LIN {X 0,Y 143.609,Z 288.097,A -85,B 0,C 180,E1 -24488.458,E2 -24488.458} C_VEL
LIN {X 0,Y 143.503,Z 288.112,A -85,B 0,C 180,E1 -24491.628,E2 -24491.628} C_VEL
LIN {X 0,Y 143.269,Z 288.273,A -85,B 0,C 180,E1 -24497.133,E2 -24497.133} C_VEL
LIN {X 0,Y 143.376,Z 289.137,A -85,B 0,C 180,E1 -24501.358,E2 -24501.358} C_VEL
LIN {X 0,Y 143.505,Z 290.831,A -85,B 0,C 180,E1 -24508.174,E2 -24508.174} C_VEL
LIN {X 0,Y 143.599,Z 291.615,A -85,B 0,C 180,E1 -24510.634,E2 -24510.634} C_VEL
LIN {X 0,Y 144.649,Z 294.631,A -85,B 0,C 180,E1 -24511.708,E2 -24511.708} C_VEL
LIN {X 0,Y 147.147,Z 297.644,A -85,B 0,C 180,E1 -24513.694,E2 -24513.694} C_VEL
LIN {X 0,Y 149.119,Z 301.806,A -85,B 0,C 180,E1 -24515.488,E2 -24515.488} C_VEL
LIN {X 0,Y 150.527,Z 303.861,A -85,B 0,C 180,E1 -24516.55,E2 -24516.55} C_VEL
LIN {X 0,Y 154.857,Z 313.083,A -85,B 0,C 180,E1 -24520.312,E2 -24520.312} C_VEL
LIN {X 0,Y 156.952,Z 319.223,A -85,B 0,C 180,E1 -24522.467,E2 -24522.467} C_VEL
LIN {X 0,Y 158.644,Z 326.853,A -85,B 0,C 180,E1 -24524.863,E2 -24524.863} C_VEL
LIN {X 0,Y 159.712,Z 336.585,A -85,B 0,C 180,E1 -24527.852,E2 -24527.852} C_VEL
LIN {X 0,Y 159.81,Z 346.242,A -85,B 0,C 180,E1 -24530.916,E2 -24530.916} C_VEL
LIN {X 0,Y 159.176,Z 354.738,A -85,B 0,C 180,E1 -24533.821,E2 -24533.821} C_VEL
LIN {X 0,Y 158.053,Z 361.316,A -85,B 0,C 180,E1 -24536.233,E2 -24536.233} C_VEL
LIN {X 0,Y 154.42,Z 369.15,A -85,B 0,C 180,E1 -24539.203,E2 -24539.203} C_VEL
LIN {X 0,Y 151.191,Z 375.693,A -85,B 0,C 180,E1 -24542.301,E2 -24542.301} C_VEL
LIN {X 0,Y 148.829,Z 380.197,A -85,B 0,C 180,E1 -24544.85,E2 -24544.85} C_VEL
LIN {X 0,Y 145.799,Z 385.692,A -85,B 0,C 180,E1 -24548.807,E2 -24548.807} C_VEL
LIN {X 0,Y 143.393,Z 390.021,A -85,B 0,C 180,E1 -24552.898,E2 -24552.898} C_VEL
LIN {X 0,Y 142.297,Z 392.395,A -85,B 0,C 180,E1 -24555.703,E2 -24555.703} C_VEL
LIN {X 0,Y 141.459,Z 394.201,A -85,B 0,C 180,E1 -24558.538,E2 -24558.538} C_VEL
LIN {X 0,Y 140.648,Z 396.664,A -85,B 0,C 180,E1 -24564.265,E2 -24564.265} C_VEL
LIN {X 0,Y 140.521,Z 397.259,A -85,B 0,C 180,E1 -24567.133,E2 -24567.133} C_VEL
LIN {X 0,Y 140.592,Z 397.419,A -85,B 0,C 180,E1 -24570,E2 -24570} C_VEL
LIN {X 0,Y 140.521,Z 397.259,A -85,B 0,C 180,E1 -24572.867,E2 -24572.867} C_VEL
LIN {X 0,Y 140.649,Z 396.664,A -85,B 0,C 180,E1 -24575.735,E2 -24575.735} C_VEL
LIN {X 0,Y 141.461,Z 394.201,A -85,B 0,C 180,E1 -24581.462,E2 -24581.462} C_VEL
LIN {X 0,Y 142.833,Z 391.242,A -85,B 0,C 180,E1 -24585.701,E2 -24585.701} C_VEL
LIN {X 0,Y 144.926,Z 387.247,A -85,B 0,C 180,E1 -24589.843,E2 -24589.843} C_VEL
LIN {X 0,Y 147.714,Z 382.113,A -85,B 0,C 180,E1 -24593.854,E2 -24593.854} C_VEL
LIN {X 0,Y 150.6,Z 376.85,A -85,B 0,C 180,E1 -24597.064,E2 -24597.064} C_VEL
LIN {X 0,Y 153.688,Z 370.526,A -85,B 0,C 180,E1 -24600.199,E2 -24600.199} C_VEL
LIN {X 0,Y 156.598,Z 364.574,A -85,B 0,C 180,E1 -24602.584,E2 -24602.584} C_VEL
LIN {X 0,Y 158.009,Z 361.314,A -85,B 0,C 180,E1 -24603.778,E2 -24603.778} C_VEL
LIN {X 0,Y 159.397,Z 352.982,A -85,B 0,C 180,E1 -24606.827,E2 -24606.827} C_VEL
LIN {X 0,Y 159.88,Z 342.962,A -85,B 0,C 180,E1 -24610.152,E2 -24610.152} C_VEL
LIN {X 0,Y 159.446,Z 333.125,A -85,B 0,C 180,E1 -24613.193,E2 -24613.193} C_VEL
LIN {X 0,Y 158.147,Z 324.133,A -85,B 0,C 180,E1 -24615.96,E2 -24615.96} C_VEL
LIN {X 0,Y 156.268,Z 316.945,A -85,B 0,C 180,E1 -24618.337,E2 -24618.337} C_VEL
LIN {X 0,Y 152.976,Z 308.875,A -85,B 0,C 180,E1 -24621.352,E2 -24621.352} C_VEL
LIN {X 0,Y 150.448,Z 303.601,A -85,B 0,C 180,E1 -24623.532,E2 -24623.532} C_VEL
LIN {X 0,Y 147.826,Z 299.371,A -85,B 0,C 180,E1 -24625.623,E2 -24625.623} C_VEL
LIN {X 0,Y 147.009,Z 297.41,A -85,B 0,C 180,E1 -24626.426,E2 -24626.426} C_VEL
LIN {X 0,Y 144.656,Z 294.581,A -85,B 0,C 180,E1 -24628.293,E2 -24628.293} C_VEL
LIN {X 0,Y 143.65,Z 291.95,A -85,B 0,C 180,E1 -24629.276,E2 -24629.276} C_VEL
LIN {X 0,Y 143.554,Z 291.417,A -85,B 0,C 180,E1 -24629.466,E2 -24629.466} C_VEL
LIN {X 0,Y 142.735,Z 290.904,A -85,B 0,C 180,E1 -24631.797,E2 -24631.797} C_VEL
LIN {X 0,Y 141.131,Z 290.55,A -85,B 0,C 180,E1 -24634.102,E2 -24634.102} C_VEL
LIN {X 0,Y 136.638,Z 289.817,A -85,B 0,C 180,E1 -24640.45,E2 -24640.45} C_VEL
LIN {X 0,Y 136.251,Z 289.554,A -85,B 0,C 180,E1 -24642.123,E2 -24642.123} C_VEL
LIN {X 0,Y 136.231,Z 289.039,A -85,B 0,C 180,E1 -24645.035,E2 -24645.035} C_VEL
LIN {X 0,Y 136.431,Z 288.991,A -85,B 0,C 180,E1 -24648.162,E2 -24648.162} C_VEL
LIN {X 0,Y 136.548,Z 288.976,A -85,B 0,C 180,E1 -24651.101,E2 -24651.101} C_VEL
LIN {X 0,Y 137.108,Z 288.873,A -85,B 0,C 180,E1 -24659.983,E2 -24659.983} C_VEL
LIN {X 0,Y 136.538,Z 288.969,A -85,B 0,C 180,E1 -24668.865,E2 -24668.865} C_VEL
LIN {X 0,Y 136.403,Z 288.993,A -85,B 0,C 180,E1 -24671.875,E2 -24671.875} C_VEL
LIN {X 0,Y 136.155,Z 289.024,A -85,B 0,C 180,E1 -24678.022,E2 -24678.022} C_VEL
LIN {X 0,Y 136.139,Z 289.023,A -85,B 0,C 180,E1 -24681.688,E2 -24681.688} C_VEL
LIN {X 0,Y 136.07,Z 289.034,A -85,B 0,C 180,E1 -24684.996,E2 -24684.996} C_VEL
LIN {X 0,Y 136.754,Z 291.283,A -85,B 0,C 180,E1 -24685.983,E2 -24685.983} C_VEL
LIN {X 0,Y 138.867,Z 293.818,A -85,B 0,C 180,E1 -24688.285,E2 -24688.285} C_VEL
LIN {X 0,Y 140.11,Z 294.726,A -85,B 0,C 180,E1 -24689.425,E2 -24689.425} C_VEL
LIN {X 0,Y 141.489,Z 297.604,A -85,B 0,C 180,E1 -24690.999,E2 -24690.999} C_VEL
LIN {X 0,Y 143.661,Z 299.964,A -85,B 0,C 180,E1 -24692.878,E2 -24692.878} C_VEL
LIN {X 0,Y 144.804,Z 302.24,A -85,B 0,C 180,E1 -24694.074,E2 -24694.074} C_VEL
LIN {X 0,Y 146.114,Z 303.884,A -85,B 0,C 180,E1 -24695.231,E2 -24695.231} C_VEL
LIN {X 0,Y 150.59,Z 311.718,A -85,B 0,C 180,E1 -24699.357,E2 -24699.357} C_VEL
LIN {X 0,Y 154.643,Z 320.363,A -85,B 0,C 180,E1 -24703.353,E2 -24703.353} C_VEL
LIN {X 0,Y 157.904,Z 329.461,A -85,B 0,C 180,E1 -24707.206,E2 -24707.206} C_VEL
LIN {X 0,Y 160.004,Z 337.281,A -85,B 0,C 180,E1 -24710.402,E2 -24710.402} C_VEL
LIN {X 0,Y 161.566,Z 346.214,A -85,B 0,C 180,E1 -24714.116,E2 -24714.116} C_VEL
LIN {X 0,Y 162.581,Z 353.438,A -85,B 0,C 180,E1 -24717.342,E2 -24717.342} C_VEL
LIN {X 0,Y 164.624,Z 361.086,A -85,B 0,C 180,E1 -24721.391,E2 -24721.391} C_VEL
LIN {X 0,Y 167.724,Z 367.177,A -85,B 0,C 180,E1 -24725.228,E2 -24725.228} C_VEL
LIN {X 0,Y 170.999,Z 371.462,A -85,B 0,C 180,E1 -24728.291,E2 -24728.291} C_VEL
LIN {X 0,Y 176.78,Z 376.47,A -85,B 0,C 180,E1 -24732.525,E2 -24732.525} C_VEL
LIN {X 0,Y 184.262,Z 380.618,A -85,B 0,C 180,E1 -24736.771,E2 -24736.771} C_VEL
LIN {X 0,Y 192.326,Z 383.551,A -85,B 0,C 180,E1 -24740.527,E2 -24740.527} C_VEL
LIN {X 0,Y 200.968,Z 385.523,A -85,B 0,C 180,E1 -24743.978,E2 -24743.978} C_VEL
LIN {X 0,Y 206.73,Z 386.382,A -85,B 0,C 180,E1 -24746.101,E2 -24746.101} C_VEL
LIN {X 0,Y 212.196,Z 386.787,A -85,B 0,C 180,E1 -24748.102,E2 -24748.102} C_VEL
LIN {X 0,Y 216.474,Z 386.827,A -85,B 0,C 180,E1 -24750,E2 -24750} C_VEL
LIN {X 0,Y 212.23,Z 386.786,A -85,B 0,C 180,E1 -24751.898,E2 -24751.898} C_VEL
LIN {X 0,Y 204.461,Z 386.098,A -85,B 0,C 180,E1 -24754.751,E2 -24754.751} C_VEL
LIN {X 0,Y 195.201,Z 384.349,A -85,B 0,C 180,E1 -24758.28,E2 -24758.28} C_VEL
LIN {X 0,Y 186.757,Z 381.669,A -85,B 0,C 180,E1 -24762.001,E2 -24762.001} C_VEL
LIN {X 0,Y 179.348,Z 378.066,A -85,B 0,C 180,E1 -24765.92,E2 -24765.92} C_VEL
LIN {X 0,Y 173.658,Z 374.035,A -85,B 0,C 180,E1 -24769.599,E2 -24769.599} C_VEL
LIN {X 0,Y 169.332,Z 369.44,A -85,B 0,C 180,E1 -24773.186,E2 -24773.186} C_VEL
LIN {X 0,Y 165.748,Z 363.566,A -85,B 0,C 180,E1 -24777.11,E2 -24777.11} C_VEL
LIN {X 0,Y 163.445,Z 357.24,A -85,B 0,C 180,E1 -24780.72,E2 -24780.72} C_VEL
LIN {X 0,Y 161.991,Z 349.766,A -85,B 0,C 180,E1 -24784.333,E2 -24784.333} C_VEL
LIN {X 0,Y 161.21,Z 343.695,A -85,B 0,C 180,E1 -24786.941,E2 -24786.941} C_VEL
LIN {X 0,Y 159.262,Z 334.483,A -85,B 0,C 180,E1 -24790.725,E2 -24790.725} C_VEL
LIN {X 0,Y 156.773,Z 326.032,A -85,B 0,C 180,E1 -24794.196,E2 -24794.196} C_VEL
LIN {X 0,Y 153.671,Z 318.238,A -85,B 0,C 180,E1 -24797.603,E2 -24797.603} C_VEL
LIN {X 0,Y 149.725,Z 310.274,A -85,B 0,C 180,E1 -24801.43,E2 -24801.43} C_VEL
LIN {X 0,Y 145.785,Z 303.546,A -85,B 0,C 180,E1 -24805.037,E2 -24805.037} C_VEL
LIN {X 0,Y 143.651,Z 300.008,A -85,B 0,C 180,E1 -24807.119,E2 -24807.119} C_VEL
LIN {X 0,Y 142.976,Z 299.168,A -85,B 0,C 180,E1 -24807.707,E2 -24807.707} C_VEL
LIN {X 0,Y 140.831,Z 296.559,A -85,B 0,C 180,E1 -24809.672,E2 -24809.672} C_VEL
LIN {X 0,Y 140.049,Z 294.565,A -85,B 0,C 180,E1 -24810.654,E2 -24810.654} C_VEL
LIN {X 0,Y 137.336,Z 292.246,A -85,B 0,C 180,E1 -24813.318,E2 -24813.318} C_VEL
LIN {X 0,Y 136.23,Z 289.93,A -85,B 0,C 180,E1 -24814.729,E2 -24814.729} C_VEL
LIN {X 0,Y 136.041,Z 289.029,A -85,B 0,C 180,E1 -24815.202,E2 -24815.202} C_VEL
LIN {X 0,Y 136.175,Z 289.015,A -85,B 0,C 180,E1 -24818.842,E2 -24818.842} C_VEL
LIN {X 0,Y 136.217,Z 289.007,A -85,B 0,C 180,E1 -24825.069,E2 -24825.069} C_VEL
LIN {X 0,Y 136.415,Z 288.991,A -85,B 0,C 180,E1 -24828.195,E2 -24828.195} C_VEL
LIN {X 0,Y 136.538,Z 288.969,A -85,B 0,C 180,E1 -24831.135,E2 -24831.135} C_VEL
LIN {X 0,Y 137.108,Z 288.873,A -85,B 0,C 180,E1 -24840.017,E2 -24840.017} C_VEL
LIN {X 0,Y 136.539,Z 288.977,A -85,B 0,C 180,E1 -24848.9,E2 -24848.9} C_VEL
LIN {X 0,Y 136.419,Z 288.995,A -85,B 0,C 180,E1 -24851.909,E2 -24851.909} C_VEL
LIN {X 0,Y 136.231,Z 289.039,A -85,B 0,C 180,E1 -24854.965,E2 -24854.965} C_VEL
LIN {X 0,Y 136.374,Z 290.211,A -85,B 0,C 180,E1 -24861.163,E2 -24861.163} C_VEL
LIN {X 0,Y 136.392,Z 291.281,A -85,B 0,C 180,E1 -24865.073,E2 -24865.073} C_VEL
LIN {X 0,Y 137.476,Z 294.259,A -85,B 0,C 180,E1 -24866.486,E2 -24866.486} C_VEL
LIN {X 0,Y 140.055,Z 297.363,A -85,B 0,C 180,E1 -24869.082,E2 -24869.082} C_VEL
LIN {X 0,Y 140.587,Z 298.2,A -85,B 0,C 180,E1 -24869.635,E2 -24869.635} C_VEL
LIN {X 0,Y 142.177,Z 301.62,A -85,B 0,C 180,E1 -24871.388,E2 -24871.388} C_VEL
LIN {X 0,Y 143.918,Z 303.998,A -85,B 0,C 180,E1 -24872.924,E2 -24872.924} C_VEL
LIN {X 0,Y 145.548,Z 307.451,A -85,B 0,C 180,E1 -24874.584,E2 -24874.584} C_VEL
LIN {X 0,Y 146.283,Z 308.544,A -85,B 0,C 180,E1 -24875.241,E2 -24875.241} C_VEL
LIN {X 0,Y 150.363,Z 318.156,A -85,B 0,C 180,E1 -24879.449,E2 -24879.449} C_VEL
LIN {X 0,Y 152.322,Z 325.052,A -85,B 0,C 180,E1 -24882.01,E2 -24882.01} C_VEL
LIN {X 0,Y 153.319,Z 332.074,A -85,B 0,C 180,E1 -24884.393,E2 -24884.393} C_VEL
LIN {X 0,Y 153.836,Z 339.832,A -85,B 0,C 180,E1 -24886.986,E2 -24886.986} C_VEL
LIN {X 0,Y 153.724,Z 347.362,A -85,B 0,C 180,E1 -24889.557,E2 -24889.557} C_VEL
LIN {X 0,Y 152.974,Z 355.099,A -85,B 0,C 180,E1 -24892.355,E2 -24892.355} C_VEL
LIN {X 0,Y 151.982,Z 361.096,A -85,B 0,C 180,E1 -24894.689,E2 -24894.689} C_VEL
LIN {X 0,Y 150.647,Z 364.362,A -85,B 0,C 180,E1 -24895.957,E2 -24895.957} C_VEL
LIN {X 0,Y 147.618,Z 370.315,A -85,B 0,C 180,E1 -24898.42,E2 -24898.42} C_VEL
LIN {X 0,Y 144.899,Z 375.481,A -85,B 0,C 180,E1 -24900.986,E2 -24900.986} C_VEL
LIN {X 0,Y 142.43,Z 379.986,A -85,B 0,C 180,E1 -24903.635,E2 -24903.635} C_VEL
LIN {X 0,Y 139.178,Z 385.48,A -85,B 0,C 180,E1 -24907.746,E2 -24907.746} C_VEL
LIN {X 0,Y 136.585,Z 389.808,A -85,B 0,C 180,E1 -24912.018,E2 -24912.018} C_VEL
LIN {X 0,Y 135.407,Z 392.183,A -85,B 0,C 180,E1 -24914.959,E2 -24914.959} C_VEL
LIN {X 0,Y 134.493,Z 393.989,A -85,B 0,C 180,E1 -24917.935,E2 -24917.935} C_VEL
LIN {X 0,Y 133.574,Z 396.453,A -85,B 0,C 180,E1 -24923.96,E2 -24923.96} C_VEL
LIN {X 0,Y 133.433,Z 397.048,A -85,B 0,C 180,E1 -24926.981,E2 -24926.981} C_VEL
LIN {X 0,Y 133.506,Z 397.208,A -85,B 0,C 180,E1 -24930,E2 -24930} C_VEL
LIN {X 0,Y 133.433,Z 397.048,A -85,B 0,C 180,E1 -24933.019,E2 -24933.019} C_VEL
LIN {X 0,Y 133.575,Z 396.453,A -85,B 0,C 180,E1 -24936.04,E2 -24936.04} C_VEL
LIN {X 0,Y 134.494,Z 393.989,A -85,B 0,C 180,E1 -24942.065,E2 -24942.065} C_VEL
LIN {X 0,Y 135.965,Z 391.029,A -85,B 0,C 180,E1 -24946.516,E2 -24946.516} C_VEL
LIN {X 0,Y 138.231,Z 387.035,A -85,B 0,C 180,E1 -24950.848,E2 -24950.848} C_VEL
LIN {X 0,Y 141.221,Z 381.901,A -85,B 0,C 180,E1 -24955.024,E2 -24955.024} C_VEL
LIN {X 0,Y 144.271,Z 376.638,A -85,B 0,C 180,E1 -24958.356,E2 -24958.356} C_VEL
LIN {X 0,Y 147.56,Z 370.313,A -85,B 0,C 180,E1 -24961.594,E2 -24961.594} C_VEL
LIN {X 0,Y 150.628,Z 364.361,A -85,B 0,C 180,E1 -24964.048,E2 -24964.048} C_VEL
LIN {X 0,Y 151.93,Z 361.094,A -85,B 0,C 180,E1 -24965.325,E2 -24965.325} C_VEL
LIN {X 0,Y 153.353,Z 352.09,A -85,B 0,C 180,E1 -24968.802,E2 -24968.802} C_VEL
LIN {X 0,Y 153.854,Z 343.276,A -85,B 0,C 180,E1 -24971.895,E2 -24971.895} C_VEL
LIN {X 0,Y 153.634,Z 334.642,A -85,B 0,C 180,E1 -24974.768,E2 -24974.768} C_VEL
LIN {X 0,Y 152.318,Z 325.064,A -85,B 0,C 180,E1 -24977.988,E2 -24977.988} C_VEL
LIN {X 0,Y 150.344,Z 318.211,A -85,B 0,C 180,E1 -24980.545,E2 -24980.545} C_VEL
LIN {X 0,Y 146.285,Z 308.46,A -85,B 0,C 180,E1 -24984.777,E2 -24984.777} C_VEL
LIN {X 0,Y 144.151,Z 304.62,A -85,B 0,C 180,E1 -24986.824,E2 -24986.824} C_VEL
LIN {X 0,Y 143.395,Z 303.067,A -85,B 0,C 180,E1 -24987.567,E2 -24987.567} C_VEL
LIN {X 0,Y 141.188,Z 299.854,A -85,B 0,C 180,E1 -24989.615,E2 -24989.615} C_VEL
LIN {X 0,Y 140.194,Z 297.359,A -85,B 0,C 180,E1 -24990.818,E2 -24990.818} C_VEL
LIN {X 0,Y 137.634,Z 294.521,A -85,B 0,C 180,E1 -24993.342,E2 -24993.342} C_VEL
LIN {X 0,Y 136.427,Z 291.563,A -85,B 0,C 180,E1 -24994.832,E2 -24994.832} C_VEL
LIN {X 0,Y 136.332,Z 291.011,A -85,B 0,C 180,E1 -24995.119,E2 -24995.119} C_VEL
LIN {X 0,Y 136.354,Z 290.191,A -85,B 0,C 180,E1 -24998.834,E2 -24998.834} C_VEL
LIN {X 0,Y 136.251,Z 289.554,A -85,B 0,C 180,E1 -25002.123,E2 -25002.123} C_VEL
LIN {X 0,Y 135.484,Z 289.308,A -85,B 0,C 180,E1 -25004.591,E2 -25004.591} C_VEL
LIN {X 0,Y 133.912,Z 289.346,A -85,B 0,C 180,E1 -25007.034,E2 -25007.034} C_VEL
LIN {X 0,Y 129.712,Z 289.828,A -85,B 0,C 180,E1 -25013.779,E2 -25013.779} C_VEL
LIN {X 0,Y 129.514,Z 289.847,A -85,B 0,C 180,E1 -25015.551,E2 -25015.551} C_VEL
LIN {X 0,Y 130.064,Z 289.748,A -85,B 0,C 180,E1 -25019.982,E2 -25019.982} C_VEL
LIN {X 0,Y 129.461,Z 289.849,A -85,B 0,C 180,E1 -25029.354,E2 -25029.354} C_VEL
LIN {X 0,Y 129.287,Z 289.881,A -85,B 0,C 180,E1 -25032.539,E2 -25032.539} C_VEL
LIN {X 0,Y 129.105,Z 289.967,A -85,B 0,C 180,E1 -25037.299,E2 -25037.299} C_VEL
LIN {X 0,Y 129.848,Z 292.328,A -85,B 0,C 180,E1 -25038.93,E2 -25038.93} C_VEL
LIN {X 0,Y 132.279,Z 295.025,A -85,B 0,C 180,E1 -25042.63,E2 -25042.63} C_VEL
LIN {X 0,Y 133.396,Z 295.75,A -85,B 0,C 180,E1 -25043.975,E2 -25043.975} C_VEL
LIN {X 0,Y 134.673,Z 298.541,A -85,B 0,C 180,E1 -25045.895,E2 -25045.895} C_VEL
LIN {X 0,Y 136.239,Z 300.245,A -85,B 0,C 180,E1 -25047.642,E2 -25047.642} C_VEL
LIN {X 0,Y 138.58,Z 303.972,A -85,B 0,C 180,E1 -25050.452,E2 -25050.452} C_VEL
LIN {X 0,Y 139.928,Z 305.471,A -85,B 0,C 180,E1 -25051.806,E2 -25051.806} C_VEL
LIN {X 0,Y 144.316,Z 313.327,A -85,B 0,C 180,E1 -25056.601,E2 -25056.601} C_VEL
LIN {X 0,Y 147.88,Z 320.664,A -85,B 0,C 180,E1 -25060.502,E2 -25060.502} C_VEL
LIN {X 0,Y 150.909,Z 328.553,A -85,B 0,C 180,E1 -25064.287,E2 -25064.287} C_VEL
LIN {X 0,Y 153.283,Z 337.095,A -85,B 0,C 180,E1 -25068.126,E2 -25068.126} C_VEL
LIN {X 0,Y 154.911,Z 345.903,A -85,B 0,C 180,E1 -25072.069,E2 -25072.069} C_VEL
LIN {X 0,Y 155.786,Z 354.23,A -85,B 0,C 180,E1 -25075.996,E2 -25075.996} C_VEL
LIN {X 0,Y 157.254,Z 361.31,A -85,B 0,C 180,E1 -25079.901,E2 -25079.901} C_VEL
LIN {X 0,Y 159.753,Z 367.44,A -85,B 0,C 180,E1 -25083.901,E2 -25083.901} C_VEL
LIN {X 0,Y 164.072,Z 373.302,A -85,B 0,C 180,E1 -25088.477,E2 -25088.477} C_VEL
LIN {X 0,Y 169.352,Z 377.735,A -85,B 0,C 180,E1 -25092.589,E2 -25092.589} C_VEL
LIN {X 0,Y 174.91,Z 380.899,A -85,B 0,C 180,E1 -25096.05,E2 -25096.05} C_VEL
LIN {X 0,Y 180.125,Z 383.033,A -85,B 0,C 180,E1 -25098.75,E2 -25098.75} C_VEL
LIN {X 0,Y 190.926,Z 385.74,A -85,B 0,C 180,E1 -25103.513,E2 -25103.513} C_VEL
LIN {X 0,Y 197.277,Z 386.662,A -85,B 0,C 180,E1 -25105.914,E2 -25105.914} C_VEL
LIN {X 0,Y 203.847,Z 387.108,A -85,B 0,C 180,E1 -25108.314,E2 -25108.314} C_VEL
LIN {X 0,Y 208.12,Z 387.071,A -85,B 0,C 180,E1 -25110,E2 -25110} C_VEL
LIN {X 0,Y 203.098,Z 387.057,A -85,B 0,C 180,E1 -25111.983,E2 -25111.983} C_VEL
LIN {X 0,Y 197.239,Z 386.655,A -85,B 0,C 180,E1 -25114.112,E2 -25114.112} C_VEL
LIN {X 0,Y 184.95,Z 384.451,A -85,B 0,C 180,E1 -25118.995,E2 -25118.995} C_VEL
LIN {X 0,Y 179.332,Z 382.769,A -85,B 0,C 180,E1 -25121.633,E2 -25121.633} C_VEL
LIN {X 0,Y 172.442,Z 379.67,A -85,B 0,C 180,E1 -25125.443,E2 -25125.443} C_VEL
LIN {X 0,Y 165.11,Z 374.402,A -85,B 0,C 180,E1 -25130.588,E2 -25130.588} C_VEL
LIN {X 0,Y 160.912,Z 369.192,A -85,B 0,C 180,E1 -25134.795,E2 -25134.795} C_VEL
LIN {X 0,Y 158.355,Z 364.34,A -85,B 0,C 180,E1 -25138.205,E2 -25138.205} C_VEL
LIN {X 0,Y 156.439,Z 357.773,A -85,B 0,C 180,E1 -25142.118,E2 -25142.118} C_VEL
LIN {X 0,Y 155.462,Z 350.999,A -85,B 0,C 180,E1 -25145.569,E2 -25145.569} C_VEL
LIN {X 0,Y 154.741,Z 344.625,A -85,B 0,C 180,E1 -25148.506,E2 -25148.506} C_VEL
LIN {X 0,Y 152.814,Z 335.311,A -85,B 0,C 180,E1 -25152.647,E2 -25152.647} C_VEL
LIN {X 0,Y 150.398,Z 327.156,A -85,B 0,C 180,E1 -25156.348,E2 -25156.348} C_VEL
LIN {X 0,Y 147.032,Z 318.853,A -85,B 0,C 180,E1 -25160.433,E2 -25160.433} C_VEL
LIN {X 0,Y 143.683,Z 312.226,A -85,B 0,C 180,E1 -25164.081,E2 -25164.081} C_VEL
LIN {X 0,Y 139.934,Z 305.448,A -85,B 0,C 180,E1 -25168.195,E2 -25168.195} C_VEL
LIN {X 0,Y 138.54,Z 303.944,A -85,B 0,C 180,E1 -25169.585,E2 -25169.585} C_VEL
LIN {X 0,Y 136.077,Z 300.076,A -85,B 0,C 180,E1 -25172.531,E2 -25172.531} C_VEL
LIN {X 0,Y 133.999,Z 297.417,A -85,B 0,C 180,E1 -25175.006,E2 -25175.006} C_VEL
LIN {X 0,Y 133.186,Z 295.525,A -85,B 0,C 180,E1 -25176.295,E2 -25176.295} C_VEL
LIN {X 0,Y 130.378,Z 293.154,A -85,B 0,C 180,E1 -25180.127,E2 -25180.127} C_VEL
LIN {X 0,Y 129.348,Z 290.98,A -85,B 0,C 180,E1 -25182.122,E2 -25182.122} C_VEL
LIN {X 0,Y 129.113,Z 289.902,A -85,B 0,C 180,E1 -25182.804,E2 -25182.804} C_VEL
LIN {X 0,Y 129.333,Z 289.875,A -85,B 0,C 180,E1 -25187.988,E2 -25187.988} C_VEL
LIN {X 0,Y 129.461,Z 289.849,A -85,B 0,C 180,E1 -25190.646,E2 -25190.646} C_VEL
LIN {X 0,Y 130.064,Z 289.748,A -85,B 0,C 180,E1 -25200.018,E2 -25200.018} C_VEL
LIN {X 0,Y 129.465,Z 289.86,A -85,B 0,C 180,E1 -25209.39,E2 -25209.39} C_VEL
LIN {X 0,Y 129.303,Z 289.88,A -85,B 0,C 180,E1 -25212.575,E2 -25212.575} C_VEL
LIN {X 0,Y 129.253,Z 290.767,A -85,B 0,C 180,E1 -25217.113,E2 -25217.113} C_VEL
LIN {X 0,Y 130.478,Z 293.968,A -85,B 0,C 180,E1 -25219.486,E2 -25219.486} C_VEL
LIN {X 0,Y 133.716,Z 297.729,A -85,B 0,C 180,E1 -25223.952,E2 -25223.952} C_VEL
LIN {X 0,Y 135.256,Z 301.356,A -85,B 0,C 180,E1 -25226.228,E2 -25226.228} C_VEL
LIN {X 0,Y 137.325,Z 304.012,A -85,B 0,C 180,E1 -25228.481,E2 -25228.481} C_VEL
LIN {X 0,Y 138.841,Z 307.408,A -85,B 0,C 180,E1 -25230.428,E2 -25230.428} C_VEL
LIN {X 0,Y 140.016,Z 309.061,A -85,B 0,C 180,E1 -25231.654,E2 -25231.654} C_VEL
LIN {X 0,Y 142.981,Z 315.704,A -85,B 0,C 180,E1 -25235.097,E2 -25235.097} C_VEL
LIN {X 0,Y 145.866,Z 323.593,A -85,B 0,C 180,E1 -25238.799,E2 -25238.799} C_VEL
LIN {X 0,Y 147.273,Z 329.995,A -85,B 0,C 180,E1 -25241.372,E2 -25241.372} C_VEL
LIN {X 0,Y 147.871,Z 337.781,A -85,B 0,C 180,E1 -25244.152,E2 -25244.152} C_VEL
LIN {X 0,Y 147.835,Z 346.044,A -85,B 0,C 180,E1 -25247.148,E2 -25247.148} C_VEL
LIN {X 0,Y 147.215,Z 353.163,A -85,B 0,C 180,E1 -25249.824,E2 -25249.824} C_VEL
LIN {X 0,Y 145.902,Z 360.872,A -85,B 0,C 180,E1 -25252.979,E2 -25252.979} C_VEL
LIN {X 0,Y 144.787,Z 364.149,A -85,B 0,C 180,E1 -25254.375,E2 -25254.375} C_VEL
LIN {X 0,Y 141.579,Z 370.103,A -85,B 0,C 180,E1 -25256.905,E2 -25256.905} C_VEL
LIN {X 0,Y 138.168,Z 376.159,A -85,B 0,C 180,E1 -25260.076,E2 -25260.076} C_VEL
LIN {X 0,Y 136.103,Z 379.775,A -85,B 0,C 180,E1 -25262.307,E2 -25262.307} C_VEL
LIN {X 0,Y 132.609,Z 385.268,A -85,B 0,C 180,E1 -25266.579,E2 -25266.579} C_VEL
LIN {X 0,Y 129.815,Z 389.596,A -85,B 0,C 180,E1 -25271.045,E2 -25271.045} C_VEL
LIN {X 0,Y 128.544,Z 391.971,A -85,B 0,C 180,E1 -25274.135,E2 -25274.135} C_VEL
LIN {X 0,Y 127.522,Z 393.777,A -85,B 0,C 180,E1 -25277.265,E2 -25277.265} C_VEL
LIN {X 0,Y 126.495,Z 396.241,A -85,B 0,C 180,E1 -25283.62,E2 -25283.62} C_VEL
LIN {X 0,Y 126.34,Z 396.837,A -85,B 0,C 180,E1 -25286.811,E2 -25286.811} C_VEL
LIN {X 0,Y 126.422,Z 396.997,A -85,B 0,C 180,E1 -25290,E2 -25290} C_VEL
LIN {X 0,Y 126.34,Z 396.837,A -85,B 0,C 180,E1 -25293.189,E2 -25293.189} C_VEL
LIN {X 0,Y 126.496,Z 396.241,A -85,B 0,C 180,E1 -25296.38,E2 -25296.38} C_VEL
LIN {X 0,Y 127.523,Z 393.777,A -85,B 0,C 180,E1 -25302.735,E2 -25302.735} C_VEL
LIN {X 0,Y 129.137,Z 390.817,A -85,B 0,C 180,E1 -25307.417,E2 -25307.417} C_VEL
LIN {X 0,Y 131.591,Z 386.823,A -85,B 0,C 180,E1 -25311.953,E2 -25311.953} C_VEL
LIN {X 0,Y 134.801,Z 381.689,A -85,B 0,C 180,E1 -25316.305,E2 -25316.305} C_VEL
LIN {X 0,Y 137.376,Z 377.582,A -85,B 0,C 180,E1 -25319.078,E2 -25319.078} C_VEL
LIN {X 0,Y 140.718,Z 371.616,A -85,B 0,C 180,E1 -25322.387,E2 -25322.387} C_VEL
LIN {X 0,Y 143.945,Z 365.776,A -85,B 0,C 180,E1 -25325.007,E2 -25325.007} C_VEL
LIN {X 0,Y 145.426,Z 362.514,A -85,B 0,C 180,E1 -25326.299,E2 -25326.299} C_VEL
LIN {X 0,Y 146.792,Z 356.036,A -85,B 0,C 180,E1 -25328.999,E2 -25328.999} C_VEL
LIN {X 0,Y 147.651,Z 348.87,A -85,B 0,C 180,E1 -25331.787,E2 -25331.787} C_VEL
LIN {X 0,Y 147.987,Z 341.341,A -85,B 0,C 180,E1 -25334.554,E2 -25334.554} C_VEL
LIN {X 0,Y 147.593,Z 332.815,A -85,B 0,C 180,E1 -25337.623,E2 -25337.623} C_VEL
LIN {X 0,Y 146.41,Z 325.59,A -85,B 0,C 180,E1 -25340.398,E2 -25340.398} C_VEL
LIN {X 0,Y 144.223,Z 318.855,A -85,B 0,C 180,E1 -25343.331,E2 -25343.331} C_VEL
LIN {X 0,Y 142.186,Z 313.663,A -85,B 0,C 180,E1 -25345.857,E2 -25345.857} C_VEL
LIN {X 0,Y 140.025,Z 309.03,A -85,B 0,C 180,E1 -25348.348,E2 -25348.348} C_VEL
LIN {X 0,Y 138.267,Z 306.32,A -85,B 0,C 180,E1 -25350.274,E2 -25350.274} C_VEL
LIN {X 0,Y 137.039,Z 303.397,A -85,B 0,C 180,E1 -25351.872,E2 -25351.872} C_VEL
LIN {X 0,Y 134.63,Z 300.257,A -85,B 0,C 180,E1 -25354.576,E2 -25354.576} C_VEL
LIN {X 0,Y 133.541,Z 297.315,A -85,B 0,C 180,E1 -25356.324,E2 -25356.324} C_VEL
LIN {X 0,Y 130.593,Z 294.17,A -85,B 0,C 180,E1 -25360.328,E2 -25360.328} C_VEL
LIN {X 0,Y 129.359,Z 291.222,A -85,B 0,C 180,E1 -25362.596,E2 -25362.596} C_VEL
LIN {X 0,Y 129.214,Z 290.494,A -85,B 0,C 180,E1 -25363.187,E2 -25363.187} C_VEL
LIN {X 0,Y 129.349,Z 289.874,A -85,B 0,C 180,E1 -25367.956,E2 -25367.956} C_VEL
LIN {X 0,Y 129.472,Z 289.859,A -85,B 0,C 180,E1 -25370.61,E2 -25370.61} C_VEL
LIN {X 0,Y 129.514,Z 289.847,A -85,B 0,C 180,E1 -25375.551,E2 -25375.551} C_VEL
LIN {X 0,Y 129.303,Z 289.986,A -85,B 0,C 180,E1 -25377.285,E2 -25377.285} C_VEL
LIN {X 0,Y 128.604,Z 290.373,A -85,B 0,C 180,E1 -25378.998,E2 -25378.998} C_VEL
LIN {X 0,Y 126.477,Z 291.631,A -85,B 0,C 180,E1 -25382.397,E2 -25382.397} C_VEL
LIN {X 0,Y 124.5,Z 293.183,A -85,B 0,C 180,E1 -25385.908,E2 -25385.908} C_VEL
LIN {X 0,Y 124.004,Z 294.266,A -85,B 0,C 180,E1 -25388.629,E2 -25388.629} C_VEL
LIN {X 0,Y 124.153,Z 294.573,A -85,B 0,C 180,E1 -25389.542,E2 -25389.542} C_VEL
LIN {X 0,Y 126.945,Z 296.876,A -85,B 0,C 180,E1 -25396.463,E2 -25396.463} C_VEL
LIN {X 0,Y 127.896,Z 299.416,A -85,B 0,C 180,E1 -25398.814,E2 -25398.814} C_VEL
LIN {X 0,Y 130.063,Z 301.696,A -85,B 0,C 180,E1 -25402.204,E2 -25402.204} C_VEL
LIN {X 0,Y 134.06,Z 307.81,A -85,B 0,C 180,E1 -25408.131,E2 -25408.131} C_VEL
LIN {X 0,Y 136.387,Z 311.347,A -85,B 0,C 180,E1 -25410.995,E2 -25410.995} C_VEL
LIN {X 0,Y 140.84,Z 320.252,A -85,B 0,C 180,E1 -25416.761,E2 -25416.761} C_VEL
LIN {X 0,Y 143.729,Z 327.344,A -85,B 0,C 180,E1 -25420.753,E2 -25420.753} C_VEL
LIN {X 0,Y 145.891,Z 334.212,A -85,B 0,C 180,E1 -25424.279,E2 -25424.279} C_VEL
LIN {X 0,Y 147.422,Z 340.639,A -85,B 0,C 180,E1 -25427.431,E2 -25427.431} C_VEL
LIN {X 0,Y 148.593,Z 348.009,A -85,B 0,C 180,E1 -25431.019,E2 -25431.019} C_VEL
LIN {X 0,Y 149.122,Z 354.244,A -85,B 0,C 180,E1 -25434.131,E2 -25434.131} C_VEL
LIN {X 0,Y 150.094,Z 361.488,A -85,B 0,C 180,E1 -25438.262,E2 -25438.262} C_VEL
LIN {X 0,Y 152.049,Z 367.697,A -85,B 0,C 180,E1 -25442.47,E2 -25442.47} C_VEL
LIN {X 0,Y 154.494,Z 371.993,A -85,B 0,C 180,E1 -25445.832,E2 -25445.832} C_VEL
LIN {X 0,Y 159.495,Z 377.237,A -85,B 0,C 180,E1 -25450.765,E2 -25450.765} C_VEL
LIN {X 0,Y 165.732,Z 381.175,A -85,B 0,C 180,E1 -25455.26,E2 -25455.26} C_VEL
LIN {X 0,Y 171.908,Z 383.709,A -85,B 0,C 180,E1 -25458.776,E2 -25458.776} C_VEL
LIN {X 0,Y 177.589,Z 385.325,A -85,B 0,C 180,E1 -25461.521,E2 -25461.521} C_VEL
LIN {X 0,Y 187.645,Z 386.946,A -85,B 0,C 180,E1 -25465.704,E2 -25465.704} C_VEL
LIN {X 0,Y 196.759,Z 387.401,A -85,B 0,C 180,E1 -25469.029,E2 -25469.029} C_VEL
LIN {X 0,Y 199.347,Z 387.327,A -85,B 0,C 180,E1 -25470,E2 -25470} C_VEL
LIN {X 0,Y 193.703,Z 387.335,A -85,B 0,C 180,E1 -25472.079,E2 -25472.079} C_VEL
LIN {X 0,Y 183.639,Z 386.411,A -85,B 0,C 180,E1 -25475.87,E2 -25475.87} C_VEL
LIN {X 0,Y 176.048,Z 384.914,A -85,B 0,C 180,E1 -25479.188,E2 -25479.188} C_VEL
LIN {X 0,Y 170.663,Z 383.321,A -85,B 0,C 180,E1 -25481.882,E2 -25481.882} C_VEL
LIN {X 0,Y 161.907,Z 379.027,A -85,B 0,C 180,E1 -25487.32,E2 -25487.32} C_VEL
LIN {X 0,Y 157.572,Z 375.616,A -85,B 0,C 180,E1 -25490.904,E2 -25490.904} C_VEL
LIN {X 0,Y 153.217,Z 369.907,A -85,B 0,C 180,E1 -25495.832,E2 -25495.832} C_VEL
LIN {X 0,Y 150.752,Z 363.987,A -85,B 0,C 180,E1 -25500.118,E2 -25500.118} C_VEL
LIN {X 0,Y 149.513,Z 358.185,A -85,B 0,C 180,E1 -25503.716,E2 -25503.716} C_VEL
LIN {X 0,Y 148.831,Z 350.25,A -85,B 0,C 180,E1 -25507.869,E2 -25507.869} C_VEL
LIN {X 0,Y 147.857,Z 343.259,A -85,B 0,C 180,E1 -25511.326,E2 -25511.326} C_VEL
LIN {X 0,Y 146.343,Z 335.853,A -85,B 0,C 180,E1 -25514.926,E2 -25514.926} C_VEL
LIN {X 0,Y 144.353,Z 329.202,A -85,B 0,C 180,E1 -25518.318,E2 -25518.318} C_VEL
LIN {X 0,Y 141.15,Z 320.983,A -85,B 0,C 180,E1 -25522.811,E2 -25522.811} C_VEL
LIN {X 0,Y 138.528,Z 315.595,A -85,B 0,C 180,E1 -25526.101,E2 -25526.101} C_VEL
LIN {X 0,Y 136.393,Z 311.33,A -85,B 0,C 180,E1 -25529.006,E2 -25529.006} C_VEL
LIN {X 0,Y 132.958,Z 306.215,A -85,B 0,C 180,E1 -25533.323,E2 -25533.323} C_VEL
LIN {X 0,Y 129.794,Z 301.49,A -85,B 0,C 180,E1 -25538.166,E2 -25538.166} C_VEL
LIN {X 0,Y 127.474,Z 298.631,A -85,B 0,C 180,E1 -25542.058,E2 -25542.058} C_VEL
LIN {X 0,Y 126.775,Z 296.589,A -85,B 0,C 180,E1 -25543.928,E2 -25543.928} C_VEL
LIN {X 0,Y 123.195,Z 291.592,A -85,B 0,C 180,E1 -25560.019,E2 -25560.019} C_VEL
LIN {X 0,Y 124.226,Z 294.671,A -85,B 0,C 180,E1 -25568.969,E2 -25568.969} C_VEL
LIN {X 0,Y 127.123,Z 297.333,A -85,B 0,C 180,E1 -25576.065,E2 -25576.065} C_VEL
LIN {X 0,Y 128.333,Z 300.757,A -85,B 0,C 180,E1 -25578.993,E2 -25578.993} C_VEL
LIN {X 0,Y 130.944,Z 303.97,A -85,B 0,C 180,E1 -25582.918,E2 -25582.918} C_VEL
LIN {X 0,Y 132.194,Z 307.266,A -85,B 0,C 180,E1 -25585.188,E2 -25585.188} C_VEL
LIN {X 0,Y 133.843,Z 309.656,A -85,B 0,C 180,E1 -25587.369,E2 -25587.369} C_VEL
LIN {X 0,Y 135.336,Z 313.213,A -85,B 0,C 180,E1 -25589.578,E2 -25589.578} C_VEL
LIN {X 0,Y 136.49,Z 315.349,A -85,B 0,C 180,E1 -25591.009,E2 -25591.009} C_VEL
LIN {X 0,Y 138.489,Z 320.43,A -85,B 0,C 180,E1 -25593.951,E2 -25593.951} C_VEL
LIN {X 0,Y 140.9,Z 327.821,A -85,B 0,C 180,E1 -25597.682,E2 -25597.682} C_VEL
LIN {X 0,Y 142.094,Z 335.067,A -85,B 0,C 180,E1 -25600.742,E2 -25600.742} C_VEL
LIN {X 0,Y 142.144,Z 344.465,A -85,B 0,C 180,E1 -25604.397,E2 -25604.397} C_VEL
LIN {X 0,Y 141.459,Z 352.489,A -85,B 0,C 180,E1 -25607.608,E2 -25607.608} C_VEL
LIN {X 0,Y 139.945,Z 360.647,A -85,B 0,C 180,E1 -25611.117,E2 -25611.117} C_VEL
LIN {X 0,Y 138.988,Z 363.935,A -85,B 0,C 180,E1 -25612.643,E2 -25612.643} C_VEL
LIN {X 0,Y 135.647,Z 369.89,A -85,B 0,C 180,E1 -25615.256,E2 -25615.256} C_VEL
LIN {X 0,Y 131.641,Z 376.559,A -85,B 0,C 180,E1 -25618.901,E2 -25618.901} C_VEL
LIN {X 0,Y 128.468,Z 381.477,A -85,B 0,C 180,E1 -25622.29,E2 -25622.29} C_VEL
LIN {X 0,Y 125.013,Z 386.611,A -85,B 0,C 180,E1 -25626.826,E2 -25626.826} C_VEL
LIN {X 0,Y 122.331,Z 390.604,A -85,B 0,C 180,E1 -25631.58,E2 -25631.58} C_VEL
LIN {X 0,Y 120.583,Z 393.565,A -85,B 0,C 180,E1 -25636.519,E2 -25636.519} C_VEL
LIN {X 0,Y 119.442,Z 396.029,A -85,B 0,C 180,E1 -25643.242,E2 -25643.242} C_VEL
LIN {X 0,Y 119.257,Z 396.625,A -85,B 0,C 180,E1 -25646.622,E2 -25646.622} C_VEL
LIN {X 0,Y 119.324,Z 396.786,A -85,B 0,C 180,E1 -25650,E2 -25650} C_VEL
LIN {X 0,Y 119.257,Z 396.625,A -85,B 0,C 180,E1 -25653.378,E2 -25653.378} C_VEL
LIN {X 0,Y 119.442,Z 396.029,A -85,B 0,C 180,E1 -25656.758,E2 -25656.758} C_VEL
LIN {X 0,Y 120.583,Z 393.565,A -85,B 0,C 180,E1 -25663.481,E2 -25663.481} C_VEL
LIN {X 0,Y 122.33,Z 390.604,A -85,B 0,C 180,E1 -25668.42,E2 -25668.42} C_VEL
LIN {X 0,Y 125.011,Z 386.611,A -85,B 0,C 180,E1 -25673.174,E2 -25673.174} C_VEL
LIN {X 0,Y 128.462,Z 381.477,A -85,B 0,C 180,E1 -25677.711,E2 -25677.711} C_VEL
LIN {X 0,Y 132.357,Z 375.397,A -85,B 0,C 180,E1 -25681.806,E2 -25681.806} C_VEL
LIN {X 0,Y 136.445,Z 368.512,A -85,B 0,C 180,E1 -25685.412,E2 -25685.412} C_VEL
LIN {X 0,Y 138.942,Z 363.933,A -85,B 0,C 180,E1 -25687.371,E2 -25687.371} C_VEL
LIN {X 0,Y 140.333,Z 358.874,A -85,B 0,C 180,E1 -25689.682,E2 -25689.682} C_VEL
LIN {X 0,Y 141.641,Z 350.632,A -85,B 0,C 180,E1 -25693.148,E2 -25693.148} C_VEL
LIN {X 0,Y 142.241,Z 341.6,A -85,B 0,C 180,E1 -25696.691,E2 -25696.691} C_VEL
LIN {X 0,Y 141.932,Z 333.401,A -85,B 0,C 180,E1 -25699.912,E2 -25699.912} C_VEL
LIN {X 0,Y 140.883,Z 327.86,A -85,B 0,C 180,E1 -25702.313,E2 -25702.313} C_VEL
LIN {X 0,Y 139.058,Z 321.934,A -85,B 0,C 180,E1 -25705.243,E2 -25705.243} C_VEL
LIN {X 0,Y 137.466,Z 317.859,A -85,B 0,C 180,E1 -25707.515,E2 -25707.515} C_VEL
LIN {X 0,Y 136.275,Z 314.578,A -85,B 0,C 180,E1 -25709.368,E2 -25709.368} C_VEL
LIN {X 0,Y 134.287,Z 310.947,A -85,B 0,C 180,E1 -25711.882,E2 -25711.882} C_VEL
LIN {X 0,Y 133.849,Z 309.636,A -85,B 0,C 180,E1 -25712.632,E2 -25712.632} C_VEL
LIN {X 0,Y 131.738,Z 306.306,A -85,B 0,C 180,E1 -25715.56,E2 -25715.56} C_VEL
LIN {X 0,Y 130.701,Z 303.527,A -85,B 0,C 180,E1 -25717.455,E2 -25717.455} C_VEL
LIN {X 0,Y 127.945,Z 299.982,A -85,B 0,C 180,E1 -25721.777,E2 -25721.777} C_VEL
LIN {X 0,Y 127.05,Z 297.122,A -85,B 0,C 180,E1 -25724.131,E2 -25724.131} C_VEL
LIN {X 0,Y 123.183,Z 291.609,A -85,B 0,C 180,E1 -25739.981,E2 -25739.981} C_VEL
LIN {X 0,Y 124.153,Z 294.573,A -85,B 0,C 180,E1 -25749.542,E2 -25749.542} C_VEL
LIN {X 0,Y 124.805,Z 296.181,A -85,B 0,C 180,E1 -25752.134,E2 -25752.134} C_VEL
LIN {X 0,Y 125.339,Z 298.869,A -85,B 0,C 180,E1 -25754.551,E2 -25754.551} C_VEL
LIN {X 0,Y 126.821,Z 307.274,A -85,B 0,C 180,E1 -25760.747,E2 -25760.747} C_VEL
LIN {X 0,Y 127.628,Z 308.839,A -85,B 0,C 180,E1 -25762.373,E2 -25762.373} C_VEL
LIN {X 0,Y 130.533,Z 313.591,A -85,B 0,C 180,E1 -25767.213,E2 -25767.213} C_VEL
LIN {X 0,Y 132.5,Z 317.066,A -85,B 0,C 180,E1 -25770.235,E2 -25770.235} C_VEL
LIN {X 0,Y 135.919,Z 324.614,A -85,B 0,C 180,E1 -25775.547,E2 -25775.547} C_VEL
LIN {X 0,Y 138.321,Z 330.905,A -85,B 0,C 180,E1 -25779.406,E2 -25779.406} C_VEL
LIN {X 0,Y 140.401,Z 338.193,A -85,B 0,C 180,E1 -25783.468,E2 -25783.468} C_VEL
LIN {X 0,Y 141.629,Z 344.573,A -85,B 0,C 180,E1 -25786.888,E2 -25786.888} C_VEL
LIN {X 0,Y 142.581,Z 353.267,A -85,B 0,C 180,E1 -25791.524,E2 -25791.524} C_VEL
LIN {X 0,Y 143.13,Z 361.785,A -85,B 0,C 180,E1 -25796.553,E2 -25796.553} C_VEL
LIN {X 0,Y 144.579,Z 368.072,A -85,B 0,C 180,E1 -25801.003,E2 -25801.003} C_VEL
LIN {X 0,Y 147.045,Z 373.066,A -85,B 0,C 180,E1 -25805.199,E2 -25805.199} C_VEL
LIN {X 0,Y 150.407,Z 377.048,A -85,B 0,C 180,E1 -25809.1,E2 -25809.1} C_VEL
LIN {X 0,Y 154.483,Z 380.273,A -85,B 0,C 180,E1 -25812.755,E2 -25812.755} C_VEL
LIN {X 0,Y 161.364,Z 383.605,A -85,B 0,C 180,E1 -25817.422,E2 -25817.422} C_VEL
LIN {X 0,Y 170.239,Z 386.048,A -85,B 0,C 180,E1 -25822.093,E2 -25822.093} C_VEL
LIN {X 0,Y 177.98,Z 387.23,A -85,B 0,C 180,E1 -25825.47,E2 -25825.47} C_VEL
LIN {X 0,Y 184.135,Z 387.619,A -85,B 0,C 180,E1 -25827.813,E2 -25827.813} C_VEL
LIN {X 0,Y 190.265,Z 387.592,A -85,B 0,C 180,E1 -25830,E2 -25830} C_VEL
LIN {X 0,Y 182.872,Z 387.541,A -85,B 0,C 180,E1 -25832.651,E2 -25832.651} C_VEL
LIN {X 0,Y 176.373,Z 387.069,A -85,B 0,C 180,E1 -25835.195,E2 -25835.195} C_VEL
LIN {X 0,Y 166.512,Z 385.196,A -85,B 0,C 180,E1 -25839.72,E2 -25839.72} C_VEL
LIN {X 0,Y 159.217,Z 382.704,A -85,B 0,C 180,E1 -25843.884,E2 -25843.884} C_VEL
LIN {X 0,Y 152.527,Z 378.893,A -85,B 0,C 180,E1 -25848.816,E2 -25848.816} C_VEL
LIN {X 0,Y 148.119,Z 374.452,A -85,B 0,C 180,E1 -25853.471,E2 -25853.471} C_VEL
LIN {X 0,Y 145.47,Z 370.162,A -85,B 0,C 180,E1 -25857.32,E2 -25857.32} C_VEL
LIN {X 0,Y 143.59,Z 364.308,A -85,B 0,C 180,E1 -25861.745,E2 -25861.745} C_VEL
LIN {X 0,Y 142.829,Z 358.76,A -85,B 0,C 180,E1 -25865.342,E2 -25865.342} C_VEL
LIN {X 0,Y 142.486,Z 351.903,A -85,B 0,C 180,E1 -25869.191,E2 -25869.191} C_VEL
LIN {X 0,Y 141.432,Z 343.582,A -85,B 0,C 180,E1 -25873.629,E2 -25873.629} C_VEL
LIN {X 0,Y 140.009,Z 336.642,A -85,B 0,C 180,E1 -25877.365,E2 -25877.365} C_VEL
LIN {X 0,Y 137.398,Z 328.32,A -85,B 0,C 180,E1 -25882.159,E2 -25882.159} C_VEL
LIN {X 0,Y 134.518,Z 321.325,A -85,B 0,C 180,E1 -25886.711,E2 -25886.711} C_VEL
LIN {X 0,Y 132.507,Z 317.048,A -85,B 0,C 180,E1 -25889.766,E2 -25889.766} C_VEL
LIN {X 0,Y 129.587,Z 312.102,A -85,B 0,C 180,E1 -25894.308,E2 -25894.308} C_VEL
LIN {X 0,Y 126.911,Z 307.757,A -85,B 0,C 180,E1 -25898.924,E2 -25898.924} C_VEL
LIN {X 0,Y 124.953,Z 304.943,A -85,B 0,C 180,E1 -25902.969,E2 -25902.969} C_VEL
LIN {X 0,Y 124.749,Z 304.294,A -85,B 0,C 180,E1 -25903.66,E2 -25903.66} C_VEL
LIN {X 0,Y 122.969,Z 302.161,A -85,B 0,C 180,E1 -25908.481,E2 -25908.481} C_VEL
LIN {X 0,Y 121.569,Z 298.631,A -85,B 0,C 180,E1 -25920.019,E2 -25920.019} C_VEL
LIN {X 0,Y 124.634,Z 303.64,A -85,B 0,C 180,E1 -25934.718,E2 -25934.718} C_VEL
LIN {X 0,Y 125.828,Z 307.207,A -85,B 0,C 180,E1 -25938.286,E2 -25938.286} C_VEL
LIN {X 0,Y 127.306,Z 309.327,A -85,B 0,C 180,E1 -25941.047,E2 -25941.047} C_VEL
LIN {X 0,Y 129.897,Z 314.677,A -85,B 0,C 180,E1 -25945.666,E2 -25945.666} C_VEL
LIN {X 0,Y 132.11,Z 319.814,A -85,B 0,C 180,E1 -25949.496,E2 -25949.496} C_VEL
LIN {X 0,Y 134.194,Z 325.702,A -85,B 0,C 180,E1 -25953.078,E2 -25953.078} C_VEL
LIN {X 0,Y 136.078,Z 332.93,A -85,B 0,C 180,E1 -25956.993,E2 -25956.993} C_VEL
LIN {X 0,Y 136.598,Z 338.343,A -85,B 0,C 180,E1 -25959.49,E2 -25959.49} C_VEL
LIN {X 0,Y 136.4,Z 345.808,A -85,B 0,C 180,E1 -25962.628,E2 -25962.628} C_VEL
LIN {X 0,Y 135.411,Z 354.03,A -85,B 0,C 180,E1 -25966.172,E2 -25966.172} C_VEL
LIN {X 0,Y 134.08,Z 360.42,A -85,B 0,C 180,E1 -25969.066,E2 -25969.066} C_VEL
LIN {X 0,Y 132.502,Z 365.351,A -85,B 0,C 180,E1 -25971.449,E2 -25971.449} C_VEL
LIN {X 0,Y 127.359,Z 373.686,A -85,B 0,C 180,E1 -25975.555,E2 -25975.555} C_VEL
LIN {X 0,Y 123.643,Z 379.35,A -85,B 0,C 180,E1 -25979.232,E2 -25979.232} C_VEL
LIN {X 0,Y 119.662,Z 384.844,A -85,B 0,C 180,E1 -25983.865,E2 -25983.865} C_VEL
LIN {X 0,Y 116.423,Z 389.172,A -85,B 0,C 180,E1 -25988.765,E2 -25988.765} C_VEL
LIN {X 0,Y 114.862,Z 391.546,A -85,B 0,C 180,E1 -25992.186,E2 -25992.186} C_VEL
LIN {X 0,Y 113.674,Z 393.353,A -85,B 0,C 180,E1 -25995.682,E2 -25995.682} C_VEL
LIN {X 0,Y 112.366,Z 395.817,A -85,B 0,C 180,E1 -26002.814,E2 -26002.814} C_VEL
LIN {X 0,Y 112.167,Z 396.414,A -85,B 0,C 180,E1 -26006.408,E2 -26006.408} C_VEL
LIN {X 0,Y 112.237,Z 396.575,A -85,B 0,C 180,E1 -26010,E2 -26010} C_VEL
LIN {X 0,Y 112.167,Z 396.414,A -85,B 0,C 180,E1 -26013.592,E2 -26013.592} C_VEL
LIN {X 0,Y 112.366,Z 395.817,A -85,B 0,C 180,E1 -26017.186,E2 -26017.186} C_VEL
LIN {X 0,Y 113.675,Z 393.353,A -85,B 0,C 180,E1 -26024.318,E2 -26024.318} C_VEL
LIN {X 0,Y 115.577,Z 390.392,A -85,B 0,C 180,E1 -26029.538,E2 -26029.538} C_VEL
LIN {X 0,Y 118.497,Z 386.399,A -85,B 0,C 180,E1 -26034.529,E2 -26034.529} C_VEL
LIN {X 0,Y 122.209,Z 381.265,A -85,B 0,C 180,E1 -26039.262,E2 -26039.262} C_VEL
LIN {X 0,Y 125.919,Z 375.808,A -85,B 0,C 180,E1 -26043.126,E2 -26043.126} C_VEL
LIN {X 0,Y 129.822,Z 369.677,A -85,B 0,C 180,E1 -26046.547,E2 -26046.547} C_VEL
LIN {X 0,Y 132.478,Z 365.35,A -85,B 0,C 180,E1 -26048.56,E2 -26048.56} C_VEL
LIN {X 0,Y 134.079,Z 360.42,A -85,B 0,C 180,E1 -26050.935,E2 -26050.935} C_VEL
LIN {X 0,Y 135.768,Z 351.809,A -85,B 0,C 180,E1 -26054.851,E2 -26054.851} C_VEL
LIN {X 0,Y 136.604,Z 342.853,A -85,B 0,C 180,E1 -26058.645,E2 -26058.645} C_VEL
LIN {X 0,Y 136.408,Z 335.556,A -85,B 0,C 180,E1 -26061.792,E2 -26061.792} C_VEL
LIN {X 0,Y 135.589,Z 330.858,A -85,B 0,C 180,E1 -26064.053,E2 -26064.053} C_VEL
LIN {X 0,Y 133.47,Z 323.503,A -85,B 0,C 180,E1 -26068.208,E2 -26068.208} C_VEL
LIN {X 0,Y 132.123,Z 319.781,A -85,B 0,C 180,E1 -26070.507,E2 -26070.507} C_VEL
LIN {X 0,Y 129.902,Z 314.663,A -85,B 0,C 180,E1 -26074.335,E2 -26074.335} C_VEL
LIN {X 0,Y 128.463,Z 312.127,A -85,B 0,C 180,E1 -26076.614,E2 -26076.614} C_VEL
LIN {X 0,Y 127.309,Z 309.319,A -85,B 0,C 180,E1 -26078.953,E2 -26078.953} C_VEL
LIN {X 0,Y 125.828,Z 307.207,A -85,B 0,C 180,E1 -26081.714,E2 -26081.714} C_VEL
LIN {X 0,Y 124.643,Z 303.603,A -85,B 0,C 180,E1 -26085.283,E2 -26085.283} C_VEL
LIN {X 0,Y 121.556,Z 298.682,A -85,B 0,C 180,E1 -26099.981,E2 -26099.981} C_VEL
LIN {X 0,Y 123.54,Z 302.698,A -85,B 0,C 180,E1 -26113.133,E2 -26113.133} C_VEL
LIN {X 0,Y 124.749,Z 304.294,A -85,B 0,C 180,E1 -26116.34,E2 -26116.34} C_VEL
LIN {X 0,Y 127.628,Z 308.839,A -85,B 0,C 180,E1 -26122.373,E2 -26122.373} C_VEL
LIN {X 0,Y 128.802,Z 311.486,A -85,B 0,C 180,E1 -26124.666,E2 -26124.666} C_VEL
LIN {X 0,Y 129.334,Z 315.094,A -85,B 0,C 180,E1 -26126.756,E2 -26126.756} C_VEL
LIN {X 0,Y 129.989,Z 325.815,A -85,B 0,C 180,E1 -26132.098,E2 -26132.098} C_VEL
LIN {X 0,Y 130.608,Z 328.048,A -85,B 0,C 180,E1 -26133.552,E2 -26133.552} C_VEL
LIN {X 0,Y 132.536,Z 333.367,A -85,B 0,C 180,E1 -26137.308,E2 -26137.308} C_VEL
LIN {X 0,Y 134.208,Z 339.352,A -85,B 0,C 180,E1 -26141.058,E2 -26141.058} C_VEL
LIN {X 0,Y 135.544,Z 346.808,A -85,B 0,C 180,E1 -26145.446,E2 -26145.446} C_VEL
LIN {X 0,Y 136.19,Z 354.143,A -85,B 0,C 180,E1 -26149.73,E2 -26149.73} C_VEL
LIN {X 0,Y 136.313,Z 361.898,A -85,B 0,C 180,E1 -26154.549,E2 -26154.549} C_VEL
LIN {X 0,Y 137.213,Z 368.202,A -85,B 0,C 180,E1 -26159.19,E2 -26159.19} C_VEL
LIN {X 0,Y 138.748,Z 372.512,A -85,B 0,C 180,E1 -26162.879,E2 -26162.879} C_VEL
LIN {X 0,Y 142.168,Z 377.427,A -85,B 0,C 180,E1 -26167.943,E2 -26167.943} C_VEL
LIN {X 0,Y 147.727,Z 381.728,A -85,B 0,C 180,E1 -26173.415,E2 -26173.415} C_VEL
LIN {X 0,Y 152.096,Z 383.887,A -85,B 0,C 180,E1 -26176.642,E2 -26176.642} C_VEL
LIN {X 0,Y 157.095,Z 385.484,A -85,B 0,C 180,E1 -26179.704,E2 -26179.704} C_VEL
LIN {X 0,Y 169.132,Z 387.564,A -85,B 0,C 180,E1 -26185.544,E2 -26185.544} C_VEL
LIN {X 0,Y 175.738,Z 387.965,A -85,B 0,C 180,E1 -26188.166,E2 -26188.166} C_VEL
LIN {X 0,Y 180.787,Z 387.869,A -85,B 0,C 180,E1 -26190,E2 -26190} C_VEL
LIN {X 0,Y 174.488,Z 387.903,A -85,B 0,C 180,E1 -26192.308,E2 -26192.308} C_VEL
LIN {X 0,Y 168.348,Z 387.513,A -85,B 0,C 180,E1 -26194.789,E2 -26194.789} C_VEL
LIN {X 0,Y 157.072,Z 385.476,A -85,B 0,C 180,E1 -26200.31,E2 -26200.31} C_VEL
LIN {X 0,Y 149.824,Z 382.843,A -85,B 0,C 180,E1 -26204.949,E2 -26204.949} C_VEL
LIN {X 0,Y 145.662,Z 380.515,A -85,B 0,C 180,E1 -26208.362,E2 -26208.362} C_VEL
LIN {X 0,Y 141.095,Z 376.145,A -85,B 0,C 180,E1 -26213.483,E2 -26213.483} C_VEL
LIN {X 0,Y 138.146,Z 371.021,A -85,B 0,C 180,E1 -26218.447,E2 -26218.447} C_VEL
LIN {X 0,Y 136.799,Z 365.884,A -85,B 0,C 180,E1 -26222.644,E2 -26222.644} C_VEL
LIN {X 0,Y 136.262,Z 359.043,A -85,B 0,C 180,E1 -26227.301,E2 -26227.301} C_VEL
LIN {X 0,Y 136.077,Z 352.242,A -85,B 0,C 180,E1 -26231.38,E2 -26231.38} C_VEL
LIN {X 0,Y 135.319,Z 345.16,A -85,B 0,C 180,E1 -26235.511,E2 -26235.511} C_VEL
LIN {X 0,Y 133.81,Z 337.873,A -85,B 0,C 180,E1 -26239.899,E2 -26239.899} C_VEL
LIN {X 0,Y 131.845,Z 331.284,A -85,B 0,C 180,E1 -26244.126,E2 -26244.126} C_VEL
LIN {X 0,Y 130.144,Z 326.773,A -85,B 0,C 180,E1 -26247.339,E2 -26247.339} C_VEL
LIN {X 0,Y 127.961,Z 321.705,A -85,B 0,C 180,E1 -26251.492,E2 -26251.492} C_VEL
LIN {X 0,Y 125.883,Z 317.801,A -85,B 0,C 180,E1 -26255.268,E2 -26255.268} C_VEL
LIN {X 0,Y 124.391,Z 314.852,A -85,B 0,C 180,E1 -26258.476,E2 -26258.476} C_VEL
LIN {X 0,Y 121.259,Z 309.613,A -85,B 0,C 180,E1 -26266.616,E2 -26266.616} C_VEL
LIN {X 0,Y 119.624,Z 305.593,A -85,B 0,C 180,E1 -26280.02,E2 -26280.02} C_VEL
LIN {X 0,Y 121.744,Z 309.882,A -85,B 0,C 180,E1 -26293.37,E2 -26293.37} C_VEL
LIN {X 0,Y 124.093,Z 315.225,A -85,B 0,C 180,E1 -26299.884,E2 -26299.884} C_VEL
LIN {X 0,Y 126.552,Z 321.275,A -85,B 0,C 180,E1 -26305.511,E2 -26305.511} C_VEL
LIN {X 0,Y 128.078,Z 325.347,A -85,B 0,C 180,E1 -26308.604,E2 -26308.604} C_VEL
LIN {X 0,Y 129.857,Z 331.688,A -85,B 0,C 180,E1 -26312.785,E2 -26312.785} C_VEL
LIN {X 0,Y 131.006,Z 338.072,A -85,B 0,C 180,E1 -26316.42,E2 -26316.42} C_VEL
LIN {X 0,Y 131.063,Z 343.726,A -85,B 0,C 180,E1 -26319.074,E2 -26319.074} C_VEL
LIN {X 0,Y 130.048,Z 352.572,A -85,B 0,C 180,E1 -26323.154,E2 -26323.154} C_VEL
LIN {X 0,Y 128.362,Z 360.255,A -85,B 0,C 180,E1 -26326.855,E2 -26326.855} C_VEL
LIN {X 0,Y 126.86,Z 365.133,A -85,B 0,C 180,E1 -26329.388,E2 -26329.388} C_VEL
LIN {X 0,Y 123.286,Z 370.842,A -85,B 0,C 180,E1 -26332.208,E2 -26332.208} C_VEL
LIN {X 0,Y 118.785,Z 377.352,A -85,B 0,C 180,E1 -26336.163,E2 -26336.163} C_VEL
LIN {X 0,Y 114.593,Z 382.969,A -85,B 0,C 180,E1 -26340.618,E2 -26340.618} C_VEL
LIN {X 0,Y 110.911,Z 387.719,A -85,B 0,C 180,E1 -26345.678,E2 -26345.678} C_VEL
LIN {X 0,Y 108.074,Z 391.333,A -85,B 0,C 180,E1 -26351.026,E2 -26351.026} C_VEL
LIN {X 0,Y 106.781,Z 393.141,A -85,B 0,C 180,E1 -26354.736,E2 -26354.736} C_VEL
LIN {X 0,Y 105.309,Z 395.605,A -85,B 0,C 180,E1 -26362.33,E2 -26362.33} C_VEL
LIN {X 0,Y 105.077,Z 396.203,A -85,B 0,C 180,E1 -26366.165,E2 -26366.165} C_VEL
LIN {X 0,Y 105.142,Z 396.364,A -85,B 0,C 180,E1 -26370,E2 -26370} C_VEL
LIN {X 0,Y 105.077,Z 396.203,A -85,B 0,C 180,E1 -26373.835,E2 -26373.835} C_VEL
LIN {X 0,Y 105.31,Z 395.605,A -85,B 0,C 180,E1 -26377.67,E2 -26377.67} C_VEL
LIN {X 0,Y 106.781,Z 393.141,A -85,B 0,C 180,E1 -26385.264,E2 -26385.264} C_VEL
LIN {X 0,Y 108.883,Z 390.179,A -85,B 0,C 180,E1 -26390.793,E2 -26390.793} C_VEL
LIN {X 0,Y 112.061,Z 386.187,A -85,B 0,C 180,E1 -26396.04,E2 -26396.04} C_VEL
LIN {X 0,Y 116.052,Z 381.054,A -85,B 0,C 180,E1 -26400.98,E2 -26400.98} C_VEL
LIN {X 0,Y 120.681,Z 374.629,A -85,B 0,C 180,E1 -26405.616,E2 -26405.616} C_VEL
LIN {X 0,Y 126.046,Z 366.704,A -85,B 0,C 180,E1 -26409.881,E2 -26409.881} C_VEL
LIN {X 0,Y 127.368,Z 363.487,A -85,B 0,C 180,E1 -26411.463,E2 -26411.463} C_VEL
LIN {X 0,Y 129.26,Z 356.423,A -85,B 0,C 180,E1 -26415.001,E2 -26415.001} C_VEL
LIN {X 0,Y 130.603,Z 348.76,A -85,B 0,C 180,E1 -26418.574,E2 -26418.574} C_VEL
LIN {X 0,Y 131.148,Z 341.478,A -85,B 0,C 180,E1 -26421.938,E2 -26421.938} C_VEL
LIN {X 0,Y 130.729,Z 335.794,A -85,B 0,C 180,E1 -26424.823,E2 -26424.823} C_VEL
LIN {X 0,Y 129.165,Z 329.03,A -85,B 0,C 180,E1 -26428.856,E2 -26428.856} C_VEL
LIN {X 0,Y 127.704,Z 324.506,A -85,B 0,C 180,E1 -26432.089,E2 -26432.089} C_VEL
LIN {X 0,Y 126.162,Z 320.323,A -85,B 0,C 180,E1 -26435.286,E2 -26435.286} C_VEL
LIN {X 0,Y 125.311,Z 318.78,A -85,B 0,C 180,E1 -26436.865,E2 -26436.865} C_VEL
LIN {X 0,Y 124.095,Z 315.22,A -85,B 0,C 180,E1 -26440.116,E2 -26440.116} C_VEL
LIN {X 0,Y 121.744,Z 309.882,A -85,B 0,C 180,E1 -26446.63,E2 -26446.63} C_VEL
LIN {X 0,Y 119.615,Z 305.62,A -85,B 0,C 180,E1 -26459.98,E2 -26459.98} C_VEL
LIN {X 0,Y 121.258,Z 309.617,A -85,B 0,C 180,E1 -26473.385,E2 -26473.385} C_VEL
LIN {X 0,Y 123.627,Z 313.784,A -85,B 0,C 180,E1 -26479.922,E2 -26479.922} C_VEL
LIN {X 0,Y 124.379,Z 314.882,A -85,B 0,C 180,E1 -26481.526,E2 -26481.526} C_VEL
LIN {X 0,Y 126.779,Z 319.265,A -85,B 0,C 180,E1 -26486.304,E2 -26486.304} C_VEL
LIN {X 0,Y 128.845,Z 323.773,A -85,B 0,C 180,E1 -26490.279,E2 -26490.279} C_VEL
LIN {X 0,Y 130.608,Z 328.048,A -85,B 0,C 180,E1 -26493.552,E2 -26493.552} C_VEL
LIN {X 0,Y 131.22,Z 330.249,A -85,B 0,C 180,E1 -26494.957,E2 -26494.957} C_VEL
LIN {X 0,Y 131.389,Z 334.138,A -85,B 0,C 180,E1 -26496.91,E2 -26496.91} C_VEL
LIN {X 0,Y 130.915,Z 338.352,A -85,B 0,C 180,E1 -26498.748,E2 -26498.748} C_VEL
LIN {X 0,Y 129.447,Z 347.428,A -85,B 0,C 180,E1 -26502.933,E2 -26502.933} C_VEL
LIN {X 0,Y 129.466,Z 349.169,A -85,B 0,C 180,E1 -26504.014,E2 -26504.014} C_VEL
LIN {X 0,Y 129.827,Z 354.563,A -85,B 0,C 180,E1 -26507.419,E2 -26507.419} C_VEL
LIN {X 0,Y 129.874,Z 360.799,A -85,B 0,C 180,E1 -26511.516,E2 -26511.516} C_VEL
LIN {X 0,Y 129.973,Z 366.685,A -85,B 0,C 180,E1 -26515.816,E2 -26515.816} C_VEL
LIN {X 0,Y 131.204,Z 372.767,A -85,B 0,C 180,E1 -26521.179,E2 -26521.179} C_VEL
LIN {X 0,Y 134.24,Z 377.972,A -85,B 0,C 180,E1 -26526.881,E2 -26526.881} C_VEL
LIN {X 0,Y 138.992,Z 382,A -85,B 0,C 180,E1 -26532.339,E2 -26532.339} C_VEL
LIN {X 0,Y 144.346,Z 384.64,A -85,B 0,C 180,E1 -26536.763,E2 -26536.763} C_VEL
LIN {X 0,Y 149.709,Z 386.33,A -85,B 0,C 180,E1 -26540.232,E2 -26540.232} C_VEL
LIN {X 0,Y 158.734,Z 387.796,A -85,B 0,C 180,E1 -26544.92,E2 -26544.92} C_VEL
LIN {X 0,Y 168.644,Z 388.224,A -85,B 0,C 180,E1 -26549.052,E2 -26549.052} C_VEL
LIN {X 0,Y 171.176,Z 388.15,A -85,B 0,C 180,E1 -26550,E2 -26550} C_VEL
LIN {X 0,Y 161.922,Z 388.003,A -85,B 0,C 180,E1 -26553.655,E2 -26553.655} C_VEL
LIN {X 0,Y 152.984,Z 386.941,A -85,B 0,C 180,E1 -26557.921,E2 -26557.921} C_VEL
LIN {X 0,Y 147.742,Z 385.758,A -85,B 0,C 180,E1 -26560.969,E2 -26560.969} C_VEL
LIN {X 0,Y 143.008,Z 384.166,A -85,B 0,C 180,E1 -26564.224,E2 -26564.224} C_VEL
LIN {X 0,Y 137.253,Z 380.859,A -85,B 0,C 180,E1 -26569.44,E2 -26569.44} C_VEL
LIN {X 0,Y 132.627,Z 375.653,A -85,B 0,C 180,E1 -26575.779,E2 -26575.779} C_VEL
LIN {X 0,Y 130.63,Z 370.796,A -85,B 0,C 180,E1 -26580.633,E2 -26580.633} C_VEL
LIN {X 0,Y 129.844,Z 365.6,A -85,B 0,C 180,E1 -26585.01,E2 -26585.01} C_VEL
LIN {X 0,Y 129.881,Z 358.645,A -85,B 0,C 180,E1 -26589.886,E2 -26589.886} C_VEL
LIN {X 0,Y 129.755,Z 352.687,A -85,B 0,C 180,E1 -26593.779,E2 -26593.779} C_VEL
LIN {X 0,Y 129.041,Z 345.392,A -85,B 0,C 180,E1 -26598.448,E2 -26598.448} C_VEL
LIN {X 0,Y 127.422,Z 337.768,A -85,B 0,C 180,E1 -26603.661,E2 -26603.661} C_VEL
LIN {X 0,Y 125.651,Z 332.156,A -85,B 0,C 180,E1 -26607.925,E2 -26607.925} C_VEL
LIN {X 0,Y 124.099,Z 327.812,A -85,B 0,C 180,E1 -26611.622,E2 -26611.622} C_VEL
LIN {X 0,Y 122.052,Z 323.413,A -85,B 0,C 180,E1 -26616.252,E2 -26616.252} C_VEL
LIN {X 0,Y 120.822,Z 320.623,A -85,B 0,C 180,E1 -26619.595,E2 -26619.595} C_VEL
LIN {X 0,Y 118.596,Z 316.497,A -85,B 0,C 180,E1 -26626.309,E2 -26626.309} C_VEL
LIN {X 0,Y 117.237,Z 314.237,A -85,B 0,C 180,E1 -26633.135,E2 -26633.135} C_VEL
LIN {X 0,Y 117.296,Z 312.408,A -85,B 0,C 180,E1 -26640.02,E2 -26640.02} C_VEL
LIN {X 0,Y 118.203,Z 315.503,A -85,B 0,C 180,E1 -26650.294,E2 -26650.294} C_VEL
LIN {X 0,Y 119.129,Z 316.961,A -85,B 0,C 180,E1 -26653.669,E2 -26653.669} C_VEL
LIN {X 0,Y 121.133,Z 322.444,A -85,B 0,C 180,E1 -26660.391,E2 -26660.391} C_VEL
LIN {X 0,Y 122.585,Z 326.838,A -85,B 0,C 180,E1 -26664.58,E2 -26664.58} C_VEL
LIN {X 0,Y 124.389,Z 333.168,A -85,B 0,C 180,E1 -26669.535,E2 -26669.535} C_VEL
LIN {X 0,Y 125.342,Z 338.368,A -85,B 0,C 180,E1 -26673.065,E2 -26673.065} C_VEL
LIN {X 0,Y 125.765,Z 342.209,A -85,B 0,C 180,E1 -26675.316,E2 -26675.316} C_VEL
LIN {X 0,Y 125.324,Z 347.611,A -85,B 0,C 180,E1 -26678.108,E2 -26678.108} C_VEL
LIN {X 0,Y 124.601,Z 352.595,A -85,B 0,C 180,E1 -26680.579,E2 -26680.579} C_VEL
LIN {X 0,Y 122.632,Z 360.615,A -85,B 0,C 180,E1 -26684.71,E2 -26684.71} C_VEL
LIN {X 0,Y 120.603,Z 366.489,A -85,B 0,C 180,E1 -26687.922,E2 -26687.922} C_VEL
LIN {X 0,Y 114.962,Z 374.417,A -85,B 0,C 180,E1 -26692.315,E2 -26692.315} C_VEL
LIN {X 0,Y 111.599,Z 378.924,A -85,B 0,C 180,E1 -26695.475,E2 -26695.475} C_VEL
LIN {X 0,Y 107.017,Z 384.418,A -85,B 0,C 180,E1 -26700.493,E2 -26700.493} C_VEL
LIN {X 0,Y 103.287,Z 388.748,A -85,B 0,C 180,E1 -26705.905,E2 -26705.905} C_VEL
LIN {X 0,Y 101.342,Z 391.12,A -85,B 0,C 180,E1 -26709.712,E2 -26709.712} C_VEL
LIN {X 0,Y 99.904,Z 392.928,A -85,B 0,C 180,E1 -26713.657,E2 -26713.657} C_VEL
LIN {X 0,Y 98.256,Z 395.393,A -85,B 0,C 180,E1 -26721.775,E2 -26721.775} C_VEL
LIN {X 0,Y 97.983,Z 395.991,A -85,B 0,C 180,E1 -26725.887,E2 -26725.887} C_VEL
LIN {X 0,Y 98.041,Z 396.152,A -85,B 0,C 180,E1 -26730,E2 -26730} C_VEL
LIN {X 0,Y 97.983,Z 395.991,A -85,B 0,C 180,E1 -26734.113,E2 -26734.113} C_VEL
LIN {X 0,Y 98.278,Z 395.394,A -85,B 0,C 180,E1 -26738.223,E2 -26738.223} C_VEL
LIN {X 0,Y 99.905,Z 392.928,A -85,B 0,C 180,E1 -26746.343,E2 -26746.343} C_VEL
LIN {X 0,Y 102.257,Z 389.967,A -85,B 0,C 180,E1 -26752.21,E2 -26752.21} C_VEL
LIN {X 0,Y 105.711,Z 385.975,A -85,B 0,C 180,E1 -26757.734,E2 -26757.734} C_VEL
LIN {X 0,Y 110.011,Z 380.842,A -85,B 0,C 180,E1 -26762.889,E2 -26762.889} C_VEL
LIN {X 0,Y 114.179,Z 375.423,A -85,B 0,C 180,E1 -26767.022,E2 -26767.022} C_VEL
LIN {X 0,Y 118.672,Z 369.252,A -85,B 0,C 180,E1 -26770.65,E2 -26770.65} C_VEL
LIN {X 0,Y 120.581,Z 366.488,A -85,B 0,C 180,E1 -26772.087,E2 -26772.087} C_VEL
LIN {X 0,Y 123.088,Z 359.148,A -85,B 0,C 180,E1 -26776.101,E2 -26776.101} C_VEL
LIN {X 0,Y 125.052,Z 350.233,A -85,B 0,C 180,E1 -26780.593,E2 -26780.593} C_VEL
LIN {X 0,Y 125.744,Z 343.471,A -85,B 0,C 180,E1 -26784.012,E2 -26784.012} C_VEL
LIN {X 0,Y 125.343,Z 338.368,A -85,B 0,C 180,E1 -26786.935,E2 -26786.935} C_VEL
LIN {X 0,Y 124.389,Z 333.21,A -85,B 0,C 180,E1 -26790.444,E2 -26790.444} C_VEL
LIN {X 0,Y 122.83,Z 327.908,A -85,B 0,C 180,E1 -26794.568,E2 -26794.568} C_VEL
LIN {X 0,Y 122.297,Z 325.911,A -85,B 0,C 180,E1 -26796.261,E2 -26796.261} C_VEL
LIN {X 0,Y 120.525,Z 320.959,A -85,B 0,C 180,E1 -26801.275,E2 -26801.275} C_VEL
LIN {X 0,Y 119.129,Z 316.961,A -85,B 0,C 180,E1 -26806.331,E2 -26806.331} C_VEL
LIN {X 0,Y 118.206,Z 315.497,A -85,B 0,C 180,E1 -26809.706,E2 -26809.706} C_VEL
LIN {X 0,Y 117.292,Z 312.419,A -85,B 0,C 180,E1 -26819.98,E2 -26819.98} C_VEL
LIN {X 0,Y 117.783,Z 315.191,A -85,B 0,C 180,E1 -26830.291,E2 -26830.291} C_VEL
LIN {X 0,Y 119.05,Z 317.405,A -85,B 0,C 180,E1 -26835.384,E2 -26835.384} C_VEL
LIN {X 0,Y 120.809,Z 320.655,A -85,B 0,C 180,E1 -26840.407,E2 -26840.407} C_VEL
LIN {X 0,Y 122.781,Z 324.8,A -85,B 0,C 180,E1 -26845.4,E2 -26845.4} C_VEL
LIN {X 0,Y 124.519,Z 328.997,A -85,B 0,C 180,E1 -26849.372,E2 -26849.372} C_VEL
LIN {X 0,Y 126.694,Z 335.403,A -85,B 0,C 180,E1 -26854.627,E2 -26854.627} C_VEL
LIN {X 0,Y 128.208,Z 341.229,A -85,B 0,C 180,E1 -26858.796,E2 -26858.796} C_VEL
LIN {X 0,Y 129.295,Z 347.627,A -85,B 0,C 180,E1 -26862.992,E2 -26862.992} C_VEL
LIN {X 0,Y 129.466,Z 349.169,A -85,B 0,C 180,E1 -26864.014,E2 -26864.014} C_VEL
LIN {X 0,Y 129.35,Z 351.621,A -85,B 0,C 180,E1 -26865.412,E2 -26865.412} C_VEL
LIN {X 0,Y 128.715,Z 354.259,A -85,B 0,C 180,E1 -26866.726,E2 -26866.726} C_VEL
LIN {X 0,Y 126.558,Z 359.407,A -85,B 0,C 180,E1 -26869.267,E2 -26869.267} C_VEL
LIN {X 0,Y 123.84,Z 365.446,A -85,B 0,C 180,E1 -26872.692,E2 -26872.692} C_VEL
LIN {X 0,Y 123.253,Z 368.477,A -85,B 0,C 180,E1 -26875.042,E2 -26875.042} C_VEL
LIN {X 0,Y 123.871,Z 373.018,A -85,B 0,C 180,E1 -26879.295,E2 -26879.295} C_VEL
LIN {X 0,Y 126.279,Z 378.361,A -85,B 0,C 180,E1 -26885.482,E2 -26885.482} C_VEL
LIN {X 0,Y 130.423,Z 382.269,A -85,B 0,C 180,E1 -26891.137,E2 -26891.137} C_VEL
LIN {X 0,Y 134.125,Z 384.439,A -85,B 0,C 180,E1 -26894.812,E2 -26894.812} C_VEL
LIN {X 0,Y 142.329,Z 387.001,A -85,B 0,C 180,E1 -26900.83,E2 -26900.83} C_VEL
LIN {X 0,Y 149.121,Z 388.081,A -85,B 0,C 180,E1 -26904.591,E2 -26904.591} C_VEL
LIN {X 0,Y 155.152,Z 388.47,A -85,B 0,C 180,E1 -26907.404,E2 -26907.404} C_VEL
LIN {X 0,Y 161.539,Z 388.431,A -85,B 0,C 180,E1 -26910,E2 -26910} C_VEL
LIN {X 0,Y 154.748,Z 388.443,A -85,B 0,C 180,E1 -26912.78,E2 -26912.78} C_VEL
LIN {X 0,Y 148.303,Z 388.02,A -85,B 0,C 180,E1 -26915.823,E2 -26915.823} C_VEL
LIN {X 0,Y 138.468,Z 386.04,A -85,B 0,C 180,E1 -26921.713,E2 -26921.713} C_VEL
LIN {X 0,Y 132.188,Z 383.437,A -85,B 0,C 180,E1 -26926.935,E2 -26926.935} C_VEL
LIN {X 0,Y 127.464,Z 379.69,A -85,B 0,C 180,E1 -26932.703,E2 -26932.703} C_VEL
LIN {X 0,Y 125.271,Z 376.665,A -85,B 0,C 180,E1 -26936.667,E2 -26936.667} C_VEL
LIN {X 0,Y 123.468,Z 370.785,A -85,B 0,C 180,E1 -26942.85,E2 -26942.85} C_VEL
LIN {X 0,Y 123.278,Z 364.868,A -85,B 0,C 180,E1 -26947.932,E2 -26947.932} C_VEL
LIN {X 0,Y 123.638,Z 358.836,A -85,B 0,C 180,E1 -26952.389,E2 -26952.389} C_VEL
LIN {X 0,Y 123.552,Z 352.357,A -85,B 0,C 180,E1 -26956.983,E2 -26956.983} C_VEL
LIN {X 0,Y 122.963,Z 346.754,A -85,B 0,C 180,E1 -26961.072,E2 -26961.072} C_VEL
LIN {X 0,Y 122.035,Z 341.69,A -85,B 0,C 180,E1 -26964.863,E2 -26964.863} C_VEL
LIN {X 0,Y 120.966,Z 337.374,A -85,B 0,C 180,E1 -26968.499,E2 -26968.499} C_VEL
LIN {X 0,Y 119.196,Z 331.869,A -85,B 0,C 180,E1 -26973.778,E2 -26973.778} C_VEL
LIN {X 0,Y 117.41,Z 327.559,A -85,B 0,C 180,E1 -26978.975,E2 -26978.975} C_VEL
LIN {X 0,Y 116.383,Z 325.225,A -85,B 0,C 180,E1 -26982.448,E2 -26982.448} C_VEL
LIN {X 0,Y 115.444,Z 322.744,A -85,B 0,C 180,E1 -26986.914,E2 -26986.914} C_VEL
LIN {X 0,Y 114.383,Z 320.818,A -85,B 0,C 180,E1 -26992.962,E2 -26992.962} C_VEL
LIN {X 0,Y 114.49,Z 319.019,A -85,B 0,C 180,E1 -27000.02,E2 -27000.02} C_VEL
LIN {X 0,Y 115.346,Z 322.152,A -85,B 0,C 180,E1 -27010.552,E2 -27010.552} C_VEL
LIN {X 0,Y 116.131,Z 324.386,A -85,B 0,C 180,E1 -27014.472,E2 -27014.472} C_VEL
LIN {X 0,Y 117.259,Z 327.928,A -85,B 0,C 180,E1 -27019.267,E2 -27019.267} C_VEL
LIN {X 0,Y 118.625,Z 333.33,A -85,B 0,C 180,E1 -27024.522,E2 -27024.522} C_VEL
LIN {X 0,Y 119.715,Z 338.561,A -85,B 0,C 180,E1 -27028.989,E2 -27028.989} C_VEL
LIN {X 0,Y 120.367,Z 344.03,A -85,B 0,C 180,E1 -27032.856,E2 -27032.856} C_VEL
LIN {X 0,Y 120.209,Z 347.648,A -85,B 0,C 180,E1 -27035.066,E2 -27035.066} C_VEL
LIN {X 0,Y 118.906,Z 354.528,A -85,B 0,C 180,E1 -27038.79,E2 -27038.79} C_VEL
LIN {X 0,Y 117.374,Z 360.129,A -85,B 0,C 180,E1 -27041.857,E2 -27041.857} C_VEL
LIN {X 0,Y 115.148,Z 366.266,A -85,B 0,C 180,E1 -27045.422,E2 -27045.422} C_VEL
LIN {X 0,Y 113.382,Z 369.041,A -85,B 0,C 180,E1 -27047.014,E2 -27047.014} C_VEL
LIN {X 0,Y 108.314,Z 375.526,A -85,B 0,C 180,E1 -27050.927,E2 -27050.927} C_VEL
LIN {X 0,Y 104.106,Z 380.63,A -85,B 0,C 180,E1 -27054.984,E2 -27054.984} C_VEL
LIN {X 0,Y 99.451,Z 385.762,A -85,B 0,C 180,E1 -27060.352,E2 -27060.352} C_VEL
LIN {X 0,Y 95.71,Z 389.756,A -85,B 0,C 180,E1 -27066.18,E2 -27066.18} C_VEL
LIN {X 0,Y 93.076,Z 392.716,A -85,B 0,C 180,E1 -27072.421,E2 -27072.421} C_VEL
LIN {X 0,Y 91.208,Z 395.181,A -85,B 0,C 180,E1 -27081.135,E2 -27081.135} C_VEL
LIN {X 0,Y 90.913,Z 395.78,A -85,B 0,C 180,E1 -27085.566,E2 -27085.566} C_VEL
LIN {X 0,Y 90.948,Z 395.941,A -85,B 0,C 180,E1 -27090,E2 -27090} C_VEL
LIN {X 0,Y 90.914,Z 395.78,A -85,B 0,C 180,E1 -27094.434,E2 -27094.434} C_VEL
LIN {X 0,Y 91.225,Z 395.182,A -85,B 0,C 180,E1 -27098.863,E2 -27098.863} C_VEL
LIN {X 0,Y 93.077,Z 392.716,A -85,B 0,C 180,E1 -27107.579,E2 -27107.579} C_VEL
LIN {X 0,Y 95.709,Z 389.756,A -85,B 0,C 180,E1 -27113.82,E2 -27113.82} C_VEL
LIN {X 0,Y 99.447,Z 385.762,A -85,B 0,C 180,E1 -27119.649,E2 -27119.649} C_VEL
LIN {X 0,Y 104.101,Z 380.63,A -85,B 0,C 180,E1 -27125.018,E2 -27125.018} C_VEL
LIN {X 0,Y 109.388,Z 374.204,A -85,B 0,C 180,E1 -27129.976,E2 -27129.976} C_VEL
LIN {X 0,Y 114.361,Z 367.662,A -85,B 0,C 180,E1 -27133.737,E2 -27133.737} C_VEL
LIN {X 0,Y 116.34,Z 363.032,A -85,B 0,C 180,E1 -27136.46,E2 -27136.46} C_VEL
LIN {X 0,Y 118.177,Z 357.361,A -85,B 0,C 180,E1 -27139.701,E2 -27139.701} C_VEL
LIN {X 0,Y 119.799,Z 350.475,A -85,B 0,C 180,E1 -27143.454,E2 -27143.454} C_VEL
LIN {X 0,Y 120.302,Z 346.192,A -85,B 0,C 180,E1 -27145.79,E2 -27145.79} C_VEL
LIN {X 0,Y 120.269,Z 342.44,A -85,B 0,C 180,E1 -27148.249,E2 -27148.249} C_VEL
LIN {X 0,Y 119.504,Z 337.41,A -85,B 0,C 180,E1 -27151.914,E2 -27151.914} C_VEL
LIN {X 0,Y 118.318,Z 331.986,A -85,B 0,C 180,E1 -27156.657,E2 -27156.657} C_VEL
LIN {X 0,Y 117.249,Z 327.948,A -85,B 0,C 180,E1 -27160.731,E2 -27160.731} C_VEL
LIN {X 0,Y 116.088,Z 324.019,A -85,B 0,C 180,E1 -27165.966,E2 -27165.966} C_VEL
LIN {X 0,Y 115.344,Z 322.158,A -85,B 0,C 180,E1 -27169.448,E2 -27169.448} C_VEL
LIN {X 0,Y 114.491,Z 319.017,A -85,B 0,C 180,E1 -27179.98,E2 -27179.98} C_VEL
LIN {X 0,Y 114.926,Z 321.818,A -85,B 0,C 180,E1 -27190.55,E2 -27190.55} C_VEL
LIN {X 0,Y 115.625,Z 323.208,A -85,B 0,C 180,E1 -27194.05,E2 -27194.05} C_VEL
LIN {X 0,Y 116.907,Z 326.267,A -85,B 0,C 180,E1 -27199.285,E2 -27199.285} C_VEL
LIN {X 0,Y 118.658,Z 330.277,A -85,B 0,C 180,E1 -27204.471,E2 -27204.471} C_VEL
LIN {X 0,Y 119.931,Z 334.055,A -85,B 0,C 180,E1 -27208.479,E2 -27208.479} C_VEL
LIN {X 0,Y 121.587,Z 339.71,A -85,B 0,C 180,E1 -27213.484,E2 -27213.484} C_VEL
LIN {X 0,Y 122.699,Z 345.047,A -85,B 0,C 180,E1 -27217.702,E2 -27217.702} C_VEL
LIN {X 0,Y 123.367,Z 350.658,A -85,B 0,C 180,E1 -27221.811,E2 -27221.811} C_VEL
LIN {X 0,Y 123.63,Z 356.436,A -85,B 0,C 180,E1 -27225.901,E2 -27225.901} C_VEL
LIN {X 0,Y 123.445,Z 362.584,A -85,B 0,C 180,E1 -27230.335,E2 -27230.335} C_VEL
LIN {X 0,Y 123.253,Z 368.477,A -85,B 0,C 180,E1 -27235.042,E2 -27235.042} C_VEL
LIN {X 0,Y 122.737,Z 370.512,A -85,B 0,C 180,E1 -27236.65,E2 -27236.65} C_VEL
LIN {X 0,Y 120.429,Z 373.954,A -85,B 0,C 180,E1 -27239.184,E2 -27239.184} C_VEL
LIN {X 0,Y 118.443,Z 377.095,A -85,B 0,C 180,E1 -27241.873,E2 -27241.873} C_VEL
LIN {X 0,Y 118.446,Z 378.544,A -85,B 0,C 180,E1 -27243.645,E2 -27243.645} C_VEL
LIN {X 0,Y 121.988,Z 382.535,A -85,B 0,C 180,E1 -27249.778,E2 -27249.778} C_VEL
LIN {X 0,Y 125.327,Z 384.711,A -85,B 0,C 180,E1 -27253.717,E2 -27253.717} C_VEL
LIN {X 0,Y 129.503,Z 386.357,A -85,B 0,C 180,E1 -27257.545,E2 -27257.545} C_VEL
LIN {X 0,Y 139.577,Z 388.366,A -85,B 0,C 180,E1 -27264.22,E2 -27264.22} C_VEL
LIN {X 0,Y 147.612,Z 388.839,A -85,B 0,C 180,E1 -27268.192,E2 -27268.192} C_VEL
LIN {X 0,Y 151.86,Z 388.715,A -85,B 0,C 180,E1 -27270,E2 -27270} C_VEL
LIN {X 0,Y 145.504,Z 388.757,A -85,B 0,C 180,E1 -27272.768,E2 -27272.768} C_VEL
LIN {X 0,Y 139.583,Z 388.366,A -85,B 0,C 180,E1 -27275.779,E2 -27275.779} C_VEL
LIN {X 0,Y 129.341,Z 386.318,A -85,B 0,C 180,E1 -27282.553,E2 -27282.553} C_VEL
LIN {X 0,Y 124.789,Z 384.434,A -85,B 0,C 180,E1 -27286.857,E2 -27286.857} C_VEL
LIN {X 0,Y 120.992,Z 381.698,A -85,B 0,C 180,E1 -27291.723,E2 -27291.723} C_VEL
LIN {X 0,Y 117.724,Z 376.919,A -85,B 0,C 180,E1 -27298.528,E2 -27298.528} C_VEL
LIN {X 0,Y 116.581,Z 371.164,A -85,B 0,C 180,E1 -27304.938,E2 -27304.938} C_VEL
LIN {X 0,Y 116.977,Z 365.062,A -85,B 0,C 180,E1 -27310.419,E2 -27310.419} C_VEL
LIN {X 0,Y 117.436,Z 359.376,A -85,B 0,C 180,E1 -27314.995,E2 -27314.995} C_VEL
LIN {X 0,Y 117.562,Z 354.391,A -85,B 0,C 180,E1 -27318.913,E2 -27318.913} C_VEL
LIN {X 0,Y 117.001,Z 347.891,A -85,B 0,C 180,E1 -27324.178,E2 -27324.178} C_VEL
LIN {X 0,Y 116.042,Z 342.375,A -85,B 0,C 180,E1 -27329.04,E2 -27329.04} C_VEL
LIN {X 0,Y 115.193,Z 338.732,A -85,B 0,C 180,E1 -27332.794,E2 -27332.794} C_VEL
LIN {X 0,Y 113.706,Z 334.201,A -85,B 0,C 180,E1 -27338.255,E2 -27338.255} C_VEL
LIN {X 0,Y 112.929,Z 331.768,A -85,B 0,C 180,E1 -27341.893,E2 -27341.893} C_VEL
LIN {X 0,Y 112.179,Z 329.799,A -85,B 0,C 180,E1 -27345.509,E2 -27345.509} C_VEL
LIN {X 0,Y 111.586,Z 328.203,A -85,B 0,C 180,E1 -27349.131,E2 -27349.131} C_VEL
LIN {X 0,Y 111.387,Z 325.489,A -85,B 0,C 180,E1 -27360.021,E2 -27360.021} C_VEL
LIN {X 0,Y 111.994,Z 328.717,A -85,B 0,C 180,E1 -27370.872,E2 -27370.872} C_VEL
LIN {X 0,Y 112.895,Z 332.034,A -85,B 0,C 180,E1 -27376.289,E2 -27376.289} C_VEL
LIN {X 0,Y 113.264,Z 333.348,A -85,B 0,C 180,E1 -27378.095,E2 -27378.095} C_VEL
LIN {X 0,Y 114.058,Z 338.292,A -85,B 0,C 180,E1 -27383.439,E2 -27383.439} C_VEL
LIN {X 0,Y 114.854,Z 343.442,A -85,B 0,C 180,E1 -27388.106,E2 -27388.106} C_VEL
LIN {X 0,Y 114.999,Z 348.925,A -85,B 0,C 180,E1 -27392.283,E2 -27392.283} C_VEL
LIN {X 0,Y 114.153,Z 353.244,A -85,B 0,C 180,E1 -27394.911,E2 -27394.911} C_VEL
LIN {X 0,Y 112.267,Z 359.802,A -85,B 0,C 180,E1 -27398.78,E2 -27398.78} C_VEL
LIN {X 0,Y 109.149,Z 367.442,A -85,B 0,C 180,E1 -27403.584,E2 -27403.584} C_VEL
LIN {X 0,Y 106.11,Z 371.582,A -85,B 0,C 180,E1 -27405.938,E2 -27405.938} C_VEL
LIN {X 0,Y 100.137,Z 378.498,A -85,B 0,C 180,E1 -27410.828,E2 -27410.828} C_VEL
LIN {X 0,Y 94.852,Z 383.994,A -85,B 0,C 180,E1 -27416.241,E2 -27416.241} C_VEL
LIN {X 0,Y 90.464,Z 388.324,A -85,B 0,C 180,E1 -27422.217,E2 -27422.217} C_VEL
LIN {X 0,Y 88.09,Z 390.695,A -85,B 0,C 180,E1 -27426.491,E2 -27426.491} C_VEL
LIN {X 0,Y 86.307,Z 392.504,A -85,B 0,C 180,E1 -27430.991,E2 -27430.991} C_VEL
LIN {X 0,Y 84.189,Z 394.97,A -85,B 0,C 180,E1 -27440.389,E2 -27440.389} C_VEL
LIN {X 0,Y 83.829,Z 395.568,A -85,B 0,C 180,E1 -27445.191,E2 -27445.191} C_VEL
LIN {X 0,Y 83.847,Z 395.73,A -85,B 0,C 180,E1 -27450,E2 -27450} C_VEL
LIN {X 0,Y 83.831,Z 395.568,A -85,B 0,C 180,E1 -27454.809,E2 -27454.809} C_VEL
LIN {X 0,Y 84.202,Z 394.97,A -85,B 0,C 180,E1 -27459.609,E2 -27459.609} C_VEL
LIN {X 0,Y 86.307,Z 392.504,A -85,B 0,C 180,E1 -27469.009,E2 -27469.009} C_VEL
LIN {X 0,Y 89.224,Z 389.543,A -85,B 0,C 180,E1 -27475.672,E2 -27475.672} C_VEL
LIN {X 0,Y 93.298,Z 385.549,A -85,B 0,C 180,E1 -27481.822,E2 -27481.822} C_VEL
LIN {X 0,Y 98.333,Z 380.417,A -85,B 0,C 180,E1 -27487.409,E2 -27487.409} C_VEL
LIN {X 0,Y 103.062,Z 375.097,A -85,B 0,C 180,E1 -27491.729,E2 -27491.729} C_VEL
LIN {X 0,Y 108.243,Z 368.827,A -85,B 0,C 180,E1 -27495.577,E2 -27495.577} C_VEL
LIN {X 0,Y 109.825,Z 366.038,A -85,B 0,C 180,E1 -27497.384,E2 -27497.384} C_VEL
LIN {X 0,Y 112.683,Z 358.651,A -85,B 0,C 180,E1 -27501.935,E2 -27501.935} C_VEL
LIN {X 0,Y 114.492,Z 351.925,A -85,B 0,C 180,E1 -27505.887,E2 -27505.887} C_VEL
LIN {X 0,Y 114.959,Z 348.986,A -85,B 0,C 180,E1 -27507.704,E2 -27507.704} C_VEL
LIN {X 0,Y 114.931,Z 344.913,A -85,B 0,C 180,E1 -27510.691,E2 -27510.691} C_VEL
LIN {X 0,Y 114.478,Z 340.396,A -85,B 0,C 180,E1 -27514.528,E2 -27514.528} C_VEL
LIN {X 0,Y 113.784,Z 336.632,A -85,B 0,C 180,E1 -27518.227,E2 -27518.227} C_VEL
LIN {X 0,Y 113.26,Z 333.354,A -85,B 0,C 180,E1 -27521.905,E2 -27521.905} C_VEL
LIN {X 0,Y 112.301,Z 329.598,A -85,B 0,C 180,E1 -27527.327,E2 -27527.327} C_VEL
LIN {X 0,Y 112.001,Z 328.705,A -85,B 0,C 180,E1 -27529.129,E2 -27529.129} C_VEL
LIN {X 0,Y 111.38,Z 325.502,A -85,B 0,C 180,E1 -27539.979,E2 -27539.979} C_VEL
LIN {X 0,Y 111.589,Z 328.197,A -85,B 0,C 180,E1 -27550.869,E2 -27550.869} C_VEL
LIN {X 0,Y 112.528,Z 330.79,A -85,B 0,C 180,E1 -27556.3,E2 -27556.3} C_VEL
LIN {X 0,Y 113.818,Z 334.48,A -85,B 0,C 180,E1 -27562.15,E2 -27562.15} C_VEL
LIN {X 0,Y 115.217,Z 338.693,A -85,B 0,C 180,E1 -27567.2,E2 -27567.2} C_VEL
LIN {X 0,Y 116.435,Z 344.491,A -85,B 0,C 180,E1 -27572.878,E2 -27572.878} C_VEL
LIN {X 0,Y 117.131,Z 349.071,A -85,B 0,C 180,E1 -27576.843,E2 -27576.843} C_VEL
LIN {X 0,Y 117.521,Z 354.444,A -85,B 0,C 180,E1 -27581.105,E2 -27581.105} C_VEL
LIN {X 0,Y 117.397,Z 360.551,A -85,B 0,C 180,E1 -27585.889,E2 -27585.889} C_VEL
LIN {X 0,Y 116.731,Z 367.387,A -85,B 0,C 180,E1 -27591.471,E2 -27591.471} C_VEL
LIN {X 0,Y 116.791,Z 373.399,A -85,B 0,C 180,E1 -27597.358,E2 -27597.358} C_VEL
LIN {X 0,Y 118.446,Z 378.544,A -85,B 0,C 180,E1 -27603.645,E2 -27603.645} C_VEL
LIN {X 0,Y 119.066,Z 380.593,A -85,B 0,C 180,E1 -27606.334,E2 -27606.334} C_VEL
LIN {X 0,Y 119.234,Z 384.818,A -85,B 0,C 180,E1 -27612.702,E2 -27612.702} C_VEL
LIN {X 0,Y 120.581,Z 386.474,A -85,B 0,C 180,E1 -27616.298,E2 -27616.298} C_VEL
LIN {X 0,Y 122.075,Z 387.157,A -85,B 0,C 180,E1 -27617.97,E2 -27617.97} C_VEL
LIN {X 0,Y 130.121,Z 388.649,A -85,B 0,C 180,E1 -27623.799,E2 -27623.799} C_VEL
LIN {X 0,Y 140.522,Z 389.053,A -85,B 0,C 180,E1 -27629.267,E2 -27629.267} C_VEL
LIN {X 0,Y 142.185,Z 389.003,A -85,B 0,C 180,E1 -27630,E2 -27630} C_VEL
LIN {X 0,Y 133.82,Z 388.905,A -85,B 0,C 180,E1 -27634.07,E2 -27634.07} C_VEL
LIN {X 0,Y 124.9,Z 387.786,A -85,B 0,C 180,E1 -27639.718,E2 -27639.718} C_VEL
LIN {X 0,Y 120.424,Z 386.59,A -85,B 0,C 180,E1 -27643.5,E2 -27643.5} C_VEL
LIN {X 0,Y 115.179,Z 383.921,A -85,B 0,C 180,E1 -27649.609,E2 -27649.609} C_VEL
LIN {X 0,Y 112.594,Z 381.649,A -85,B 0,C 180,E1 -27653.934,E2 -27653.934} C_VEL
LIN {X 0,Y 110.36,Z 377.171,A -85,B 0,C 180,E1 -27660.627,E2 -27660.627} C_VEL
LIN {X 0,Y 109.99,Z 371.407,A -85,B 0,C 180,E1 -27667.374,E2 -27667.374} C_VEL
LIN {X 0,Y 110.813,Z 365.531,A -85,B 0,C 180,E1 -27672.981,E2 -27672.981} C_VEL
LIN {X 0,Y 111.459,Z 359.6,A -85,B 0,C 180,E1 -27678.186,E2 -27678.186} C_VEL
LIN {X 0,Y 111.542,Z 353.908,A -85,B 0,C 180,E1 -27683.263,E2 -27683.263} C_VEL
LIN {X 0,Y 111.097,Z 348.294,A -85,B 0,C 180,E1 -27688.56,E2 -27688.56} C_VEL
LIN {X 0,Y 110.307,Z 343.666,A -85,B 0,C 180,E1 -27693.539,E2 -27693.539} C_VEL
LIN {X 0,Y 109.318,Z 339.403,A -85,B 0,C 180,E1 -27699.317,E2 -27699.317} C_VEL
LIN {X 0,Y 108.335,Z 336.123,A -85,B 0,C 180,E1 -27704.983,E2 -27704.983} C_VEL
LIN {X 0,Y 107.893,Z 334.512,A -85,B 0,C 180,E1 -27708.754,E2 -27708.754} C_VEL
LIN {X 0,Y 107.57,Z 332.595,A -85,B 0,C 180,E1 -27716.276,E2 -27716.276} C_VEL
LIN {X 0,Y 107.958,Z 331.81,A -85,B 0,C 180,E1 -27720.022,E2 -27720.022} C_VEL
LIN {X 0,Y 107.913,Z 333.767,A -85,B 0,C 180,E1 -27727.506,E2 -27727.506} C_VEL
LIN {X 0,Y 108.339,Z 335.093,A -85,B 0,C 180,E1 -27731.243,E2 -27731.243} C_VEL
LIN {X 0,Y 108.928,Z 338.533,A -85,B 0,C 180,E1 -27736.9,E2 -27736.9} C_VEL
LIN {X 0,Y 109.324,Z 341.738,A -85,B 0,C 180,E1 -27740.728,E2 -27740.728} C_VEL
LIN {X 0,Y 109.726,Z 347.483,A -85,B 0,C 180,E1 -27746.66,E2 -27746.66} C_VEL
LIN {X 0,Y 109.703,Z 351.184,A -85,B 0,C 180,E1 -27749.791,E2 -27749.791} C_VEL
LIN {X 0,Y 109.074,Z 354.385,A -85,B 0,C 180,E1 -27752.137,E2 -27752.137} C_VEL
LIN {X 0,Y 106.838,Z 360.925,A -85,B 0,C 180,E1 -27756.326,E2 -27756.326} C_VEL
LIN {X 0,Y 104.005,Z 367.214,A -85,B 0,C 180,E1 -27760.519,E2 -27760.519} C_VEL
LIN {X 0,Y 103.259,Z 368.61,A -85,B 0,C 180,E1 -27761.525,E2 -27761.525} C_VEL
LIN {X 0,Y 98.882,Z 373.78,A -85,B 0,C 180,E1 -27764.706,E2 -27764.706} C_VEL
LIN {X 0,Y 94.71,Z 378.286,A -85,B 0,C 180,E1 -27768.1,E2 -27768.1} C_VEL
LIN {X 0,Y 89.016,Z 383.781,A -85,B 0,C 180,E1 -27773.692,E2 -27773.692} C_VEL
LIN {X 0,Y 84.22,Z 388.112,A -85,B 0,C 180,E1 -27779.955,E2 -27779.955} C_VEL
LIN {X 0,Y 81.596,Z 390.483,A -85,B 0,C 180,E1 -27784.491,E2 -27784.491} C_VEL
LIN {X 0,Y 79.607,Z 392.292,A -85,B 0,C 180,E1 -27789.321,E2 -27789.321} C_VEL
LIN {X 0,Y 77.174,Z 394.758,A -85,B 0,C 180,E1 -27799.506,E2 -27799.506} C_VEL
LIN {X 0,Y 76.766,Z 395.357,A -85,B 0,C 180,E1 -27804.747,E2 -27804.747} C_VEL
LIN {X 0,Y 76.769,Z 395.519,A -85,B 0,C 180,E1 -27810,E2 -27810} C_VEL
LIN {X 0,Y 76.769,Z 395.358,A -85,B 0,C 180,E1 -27815.253,E2 -27815.253} C_VEL
LIN {X 0,Y 77.184,Z 394.758,A -85,B 0,C 180,E1 -27820.493,E2 -27820.493} C_VEL
LIN {X 0,Y 79.607,Z 392.292,A -85,B 0,C 180,E1 -27830.679,E2 -27830.679} C_VEL
LIN {X 0,Y 82.852,Z 389.331,A -85,B 0,C 180,E1 -27837.81,E2 -27837.81} C_VEL
LIN {X 0,Y 87.306,Z 385.337,A -85,B 0,C 180,E1 -27844.297,E2 -27844.297} C_VEL
LIN {X 0,Y 92.759,Z 380.204,A -85,B 0,C 180,E1 -27850.091,E2 -27850.091} C_VEL
LIN {X 0,Y 97.686,Z 375.051,A -85,B 0,C 180,E1 -27854.399,E2 -27854.399} C_VEL
LIN {X 0,Y 102.227,Z 369.992,A -85,B 0,C 180,E1 -27857.65,E2 -27857.65} C_VEL
LIN {X 0,Y 103.259,Z 368.61,A -85,B 0,C 180,E1 -27858.475,E2 -27858.475} C_VEL
LIN {X 0,Y 106.159,Z 362.565,A -85,B 0,C 180,E1 -27862.6,E2 -27862.6} C_VEL
LIN {X 0,Y 108.219,Z 357.355,A -85,B 0,C 180,E1 -27865.986,E2 -27865.986} C_VEL
LIN {X 0,Y 109.47,Z 352.652,A -85,B 0,C 180,E1 -27869.073,E2 -27869.073} C_VEL
LIN {X 0,Y 109.742,Z 348.674,A -85,B 0,C 180,E1 -27872.313,E2 -27872.313} C_VEL
LIN {X 0,Y 109.62,Z 345.358,A -85,B 0,C 180,E1 -27875.348,E2 -27875.348} C_VEL
LIN {X 0,Y 109.321,Z 341.744,A -85,B 0,C 180,E1 -27879.272,E2 -27879.272} C_VEL
LIN {X 0,Y 108.928,Z 338.532,A -85,B 0,C 180,E1 -27883.1,E2 -27883.1} C_VEL
LIN {X 0,Y 108.363,Z 335.056,A -85,B 0,C 180,E1 -27888.759,E2 -27888.759} C_VEL
LIN {X 0,Y 107.923,Z 333.75,A -85,B 0,C 180,E1 -27892.495,E2 -27892.495} C_VEL
LIN {X 0,Y 107.953,Z 331.819,A -85,B 0,C 180,E1 -27899.978,E2 -27899.978} C_VEL
LIN {X 0,Y 107.59,Z 333.453,A -85,B 0,C 180,E1 -27907.606,E2 -27907.606} C_VEL
LIN {X 0,Y 108.063,Z 335.05,A -85,B 0,C 180,E1 -27912.702,E2 -27912.702} C_VEL
LIN {X 0,Y 108.962,Z 338.186,A -85,B 0,C 180,E1 -27918.79,E2 -27918.79} C_VEL
LIN {X 0,Y 109.683,Z 340.629,A -85,B 0,C 180,E1 -27922.585,E2 -27922.585} C_VEL
LIN {X 0,Y 110.376,Z 344.104,A -85,B 0,C 180,E1 -27926.949,E2 -27926.949} C_VEL
LIN {X 0,Y 111.188,Z 349.295,A -85,B 0,C 180,E1 -27932.457,E2 -27932.457} C_VEL
LIN {X 0,Y 111.621,Z 355.089,A -85,B 0,C 180,E1 -27937.841,E2 -27937.841} C_VEL
LIN {X 0,Y 111.371,Z 360.902,A -85,B 0,C 180,E1 -27942.884,E2 -27942.884} C_VEL
LIN {X 0,Y 110.637,Z 366.862,A -85,B 0,C 180,E1 -27948.168,E2 -27948.168} C_VEL
LIN {X 0,Y 109.92,Z 373.512,A -85,B 0,C 180,E1 -27954.87,E2 -27954.87} C_VEL
LIN {X 0,Y 110.682,Z 378.432,A -85,B 0,C 180,E1 -27961.118,E2 -27961.118} C_VEL
LIN {X 0,Y 112.506,Z 381.652,A -85,B 0,C 180,E1 -27966.046,E2 -27966.046} C_VEL
LIN {X 0,Y 117.371,Z 385.288,A -85,B 0,C 180,E1 -27973.265,E2 -27973.265} C_VEL
LIN {X 0,Y 122.075,Z 387.157,A -85,B 0,C 180,E1 -27977.97,E2 -27977.97} C_VEL
LIN {X 0,Y 123.4,Z 387.79,A -85,B 0,C 180,E1 -27979.706,E2 -27979.706} C_VEL
LIN {X 0,Y 125.504,Z 389.243,A -85,B 0,C 180,E1 -27985.812,E2 -27985.812} C_VEL
LIN {X 0,Y 127.419,Z 389.337,A -85,B 0,C 180,E1 -27987.388,E2 -27987.388} C_VEL
LIN {X 0,Y 132.54,Z 389.29,A -85,B 0,C 180,E1 -27990,E2 -27990} C_VEL
LIN {X 0,Y 126.38,Z 389.327,A -85,B 0,C 180,E1 -27993.188,E2 -27993.188} C_VEL
LIN {X 0,Y 120.319,Z 388.898,A -85,B 0,C 180,E1 -27996.979,E2 -27996.979} C_VEL
LIN {X 0,Y 111.657,Z 386.859,A -85,B 0,C 180,E1 -28004.582,E2 -28004.582} C_VEL
LIN {X 0,Y 108.312,Z 385.242,A -85,B 0,C 180,E1 -28008.931,E2 -28008.931} C_VEL
LIN {X 0,Y 104.766,Z 381.905,A -85,B 0,C 180,E1 -28015.851,E2 -28015.851} C_VEL
LIN {X 0,Y 103.22,Z 377.421,A -85,B 0,C 180,E1 -28023.004,E2 -28023.004} C_VEL
LIN {X 0,Y 103.579,Z 371.75,A -85,B 0,C 180,E1 -28030.022,E2 -28030.022} C_VEL
LIN {X 0,Y 104.629,Z 367.105,A -85,B 0,C 180,E1 -28034.852,E2 -28034.852} C_VEL
LIN {X 0,Y 105.558,Z 360.997,A -85,B 0,C 180,E1 -28040.799,E2 -28040.799} C_VEL
LIN {X 0,Y 105.78,Z 355.482,A -85,B 0,C 180,E1 -28046.336,E2 -28046.336} C_VEL
LIN {X 0,Y 105.635,Z 352.169,A -85,B 0,C 180,E1 -28049.87,E2 -28049.87} C_VEL
LIN {X 0,Y 105.328,Z 348.507,A -85,B 0,C 180,E1 -28054.323,E2 -28054.323} C_VEL
LIN {X 0,Y 104.597,Z 344.365,A -85,B 0,C 180,E1 -28060.394,E2 -28060.394} C_VEL
LIN {X 0,Y 104.201,Z 342.235,A -85,B 0,C 180,E1 -28064.373,E2 -28064.373} C_VEL
LIN {X 0,Y 103.916,Z 340.62,A -85,B 0,C 180,E1 -28068.317,E2 -28068.317} C_VEL
LIN {X 0,Y 103.662,Z 338.606,A -85,B 0,C 180,E1 -28076.135,E2 -28076.135} C_VEL
LIN {X 0,Y 104.073,Z 337.824,A -85,B 0,C 180,E1 -28080.022,E2 -28080.022} C_VEL
LIN {X 0,Y 103.998,Z 339.829,A -85,B 0,C 180,E1 -28087.79,E2 -28087.79} C_VEL
LIN {X 0,Y 104.345,Z 342.083,A -85,B 0,C 180,E1 -28093.029,E2 -28093.029} C_VEL
LIN {X 0,Y 104.471,Z 343.576,A -85,B 0,C 180,E1 -28095.632,E2 -28095.632} C_VEL
LIN {X 0,Y 104.536,Z 346.644,A -85,B 0,C 180,E1 -28099.745,E2 -28099.745} C_VEL
LIN {X 0,Y 104.569,Z 351.368,A -85,B 0,C 180,E1 -28105.021,E2 -28105.021} C_VEL
LIN {X 0,Y 104.16,Z 355.235,A -85,B 0,C 180,E1 -28108.702,E2 -28108.702} C_VEL
LIN {X 0,Y 103.671,Z 357.215,A -85,B 0,C 180,E1 -28110.199,E2 -28110.199} C_VEL
LIN {X 0,Y 100.518,Z 364.464,A -85,B 0,C 180,E1 -28115.269,E2 -28115.269} C_VEL
LIN {X 0,Y 97.509,Z 369.777,A -85,B 0,C 180,E1 -28119.213,E2 -28119.213} C_VEL
LIN {X 0,Y 91.486,Z 376.111,A -85,B 0,C 180,E1 -28123.453,E2 -28123.453} C_VEL
LIN {X 0,Y 85.388,Z 381.91,A -85,B 0,C 180,E1 -28128.819,E2 -28128.819} C_VEL
LIN {X 0,Y 79.788,Z 386.658,A -85,B 0,C 180,E1 -28135.073,E2 -28135.073} C_VEL
LIN {X 0,Y 75.218,Z 390.271,A -85,B 0,C 180,E1 -28142.15,E2 -28142.15} C_VEL
LIN {X 0,Y 72.974,Z 392.079,A -85,B 0,C 180,E1 -28147.342,E2 -28147.342} C_VEL
LIN {X 0,Y 70.192,Z 394.546,A -85,B 0,C 180,E1 -28158.449,E2 -28158.449} C_VEL
LIN {X 0,Y 69.68,Z 395.146,A -85,B 0,C 180,E1 -28164.211,E2 -28164.211} C_VEL
LIN {X 0,Y 69.681,Z 395.308,A -85,B 0,C 180,E1 -28170,E2 -28170} C_VEL
LIN {X 0,Y 69.682,Z 395.146,A -85,B 0,C 180,E1 -28175.788,E2 -28175.788} C_VEL
LIN {X 0,Y 70.2,Z 394.546,A -85,B 0,C 180,E1 -28181.55,E2 -28181.55} C_VEL
LIN {X 0,Y 72.974,Z 392.079,A -85,B 0,C 180,E1 -28192.658,E2 -28192.658} C_VEL
LIN {X 0,Y 76.619,Z 389.119,A -85,B 0,C 180,E1 -28200.297,E2 -28200.297} C_VEL
LIN {X 0,Y 81.504,Z 385.124,A -85,B 0,C 180,E1 -28207.127,E2 -28207.127} C_VEL
LIN {X 0,Y 87.419,Z 379.992,A -85,B 0,C 180,E1 -28213.105,E2 -28213.105} C_VEL
LIN {X 0,Y 92.719,Z 374.839,A -85,B 0,C 180,E1 -28217.488,E2 -28217.488} C_VEL
LIN {X 0,Y 97.512,Z 369.777,A -85,B 0,C 180,E1 -28220.784,E2 -28220.784} C_VEL
LIN {X 0,Y 101.042,Z 363.335,A -85,B 0,C 180,E1 -28225.495,E2 -28225.495} C_VEL
LIN {X 0,Y 103.689,Z 357.16,A -85,B 0,C 180,E1 -28229.839,E2 -28229.839} C_VEL
LIN {X 0,Y 104.38,Z 353.579,A -85,B 0,C 180,E1 -28232.781,E2 -28232.781} C_VEL
LIN {X 0,Y 104.635,Z 350.209,A -85,B 0,C 180,E1 -28236.211,E2 -28236.211} C_VEL
LIN {X 0,Y 104.529,Z 346.587,A -85,B 0,C 180,E1 -28240.333,E2 -28240.333} C_VEL
LIN {X 0,Y 104.463,Z 343.587,A -85,B 0,C 180,E1 -28244.366,E2 -28244.366} C_VEL
LIN {X 0,Y 104.331,Z 341.324,A -85,B 0,C 180,E1 -28248.319,E2 -28248.319} C_VEL
LIN {X 0,Y 104.004,Z 339.82,A -85,B 0,C 180,E1 -28252.211,E2 -28252.211} C_VEL
LIN {X 0,Y 104.066,Z 337.834,A -85,B 0,C 180,E1 -28259.978,E2 -28259.978} C_VEL
LIN {X 0,Y 103.68,Z 339.468,A -85,B 0,C 180,E1 -28267.768,E2 -28267.768} C_VEL
LIN {X 0,Y 103.945,Z 340.581,A -85,B 0,C 180,E1 -28271.679,E2 -28271.679} C_VEL
LIN {X 0,Y 104.372,Z 343.251,A -85,B 0,C 180,E1 -28277.614,E2 -28277.614} C_VEL
LIN {X 0,Y 104.859,Z 345.433,A -85,B 0,C 180,E1 -28281.399,E2 -28281.399} C_VEL
LIN {X 0,Y 105.338,Z 348.495,A -85,B 0,C 180,E1 -28285.674,E2 -28285.674} C_VEL
LIN {X 0,Y 105.751,Z 354,A -85,B 0,C 180,E1 -28292.09,E2 -28292.09} C_VEL
LIN {X 0,Y 105.683,Z 358.751,A -85,B 0,C 180,E1 -28297.061,E2 -28297.061} C_VEL
LIN {X 0,Y 105.133,Z 363.761,A -85,B 0,C 180,E1 -28301.917,E2 -28301.917} C_VEL
LIN {X 0,Y 104.362,Z 368.312,A -85,B 0,C 180,E1 -28306.35,E2 -28306.35} C_VEL
LIN {X 0,Y 103.285,Z 373.758,A -85,B 0,C 180,E1 -28312.237,E2 -28312.237} C_VEL
LIN {X 0,Y 103.464,Z 378.998,A -85,B 0,C 180,E1 -28319.376,E2 -28319.376} C_VEL
LIN {X 0,Y 105.583,Z 383.061,A -85,B 0,C 180,E1 -28326.461,E2 -28326.461} C_VEL
LIN {X 0,Y 109.948,Z 386.108,A -85,B 0,C 180,E1 -28333.412,E2 -28333.412} C_VEL
LIN {X 0,Y 115.911,Z 388.083,A -85,B 0,C 180,E1 -28339.604,E2 -28339.604} C_VEL
LIN {X 0,Y 120.779,Z 388.929,A -85,B 0,C 180,E1 -28343.317,E2 -28343.317} C_VEL
LIN {X 0,Y 127.419,Z 389.337,A -85,B 0,C 180,E1 -28347.388,E2 -28347.388} C_VEL
LIN {X 0,Y 127.924,Z 389.429,A -85,B 0,C 180,E1 -28348.183,E2 -28348.183} C_VEL
LIN {X 0,Y 127.246,Z 389.448,A -85,B 0,C 180,E1 -28349.276,E2 -28349.276} C_VEL
LIN {X 0,Y 124.969,Z 389.526,A -85,B 0,C 180,E1 -28350.681,E2 -28350.681} C_VEL
LIN {X 0,Y 115.156,Z 389.478,A -85,B 0,C 180,E1 -28354.659,E2 -28354.659} C_VEL
LIN {X 0,Y 114.124,Z 389.409,A -85,B 0,C 180,E1 -28355.301,E2 -28355.301} C_VEL
LIN {X 0,Y 106.825,Z 388.333,A -85,B 0,C 180,E1 -28361.383,E2 -28361.383} C_VEL
LIN {X 0,Y 102.546,Z 386.91,A -85,B 0,C 180,E1 -28366.457,E2 -28366.457} C_VEL
LIN {X 0,Y 98.95,Z 384.619,A -85,B 0,C 180,E1 -28372.651,E2 -28372.651} C_VEL
LIN {X 0,Y 96.612,Z 380.715,A -85,B 0,C 180,E1 -28380.611,E2 -28380.611} C_VEL
LIN {X 0,Y 96.384,Z 376.938,A -85,B 0,C 180,E1 -28386.716,E2 -28386.716} C_VEL
LIN {X 0,Y 97.706,Z 371.16,A -85,B 0,C 180,E1 -28394.042,E2 -28394.042} C_VEL
LIN {X 0,Y 98.962,Z 366.452,A -85,B 0,C 180,E1 -28399.274,E2 -28399.274} C_VEL
LIN {X 0,Y 99.752,Z 362.065,A -85,B 0,C 180,E1 -28404.142,E2 -28404.142} C_VEL
LIN {X 0,Y 100.098,Z 357.257,A -85,B 0,C 180,E1 -28409.646,E2 -28409.646} C_VEL
LIN {X 0,Y 100.093,Z 353.109,A -85,B 0,C 180,E1 -28415.111,E2 -28415.111} C_VEL
LIN {X 0,Y 99.902,Z 350.337,A -85,B 0,C 180,E1 -28419.432,E2 -28419.432} C_VEL
LIN {X 0,Y 99.703,Z 348.204,A -85,B 0,C 180,E1 -28423.648,E2 -28423.648} C_VEL
LIN {X 0,Y 99.464,Z 346.483,A -85,B 0,C 180,E1 -28427.787,E2 -28427.787} C_VEL
LIN {X 0,Y 99.331,Z 345.187,A -85,B 0,C 180,E1 -28432.109,E2 -28432.109} C_VEL
LIN {X 0,Y 99.897,Z 343.653,A -85,B 0,C 180,E1 -28440.023,E2 -28440.023} C_VEL
LIN {X 0,Y 99.662,Z 346.065,A -85,B 0,C 180,E1 -28449.164,E2 -28449.164} C_VEL
LIN {X 0,Y 99.79,Z 347.331,A -85,B 0,C 180,E1 -28452.221,E2 -28452.221} C_VEL
LIN {X 0,Y 99.722,Z 349.882,A -85,B 0,C 180,E1 -28456.397,E2 -28456.397} C_VEL
LIN {X 0,Y 99.466,Z 352.97,A -85,B 0,C 180,E1 -28460.712,E2 -28460.712} C_VEL
LIN {X 0,Y 99.073,Z 356.885,A -85,B 0,C 180,E1 -28465.215,E2 -28465.215} C_VEL
LIN {X 0,Y 98.571,Z 358.99,A -85,B 0,C 180,E1 -28467.304,E2 -28467.304} C_VEL
LIN {X 0,Y 96.554,Z 363.289,A -85,B 0,C 180,E1 -28470.658,E2 -28470.658} C_VEL
LIN {X 0,Y 93.741,Z 368.151,A -85,B 0,C 180,E1 -28474.444,E2 -28474.444} C_VEL
LIN {X 0,Y 91.91,Z 370.943,A -85,B 0,C 180,E1 -28476.594,E2 -28476.594} C_VEL
LIN {X 0,Y 84.449,Z 378.01,A -85,B 0,C 180,E1 -28481.776,E2 -28481.776} C_VEL
LIN {X 0,Y 78.001,Z 383.358,A -85,B 0,C 180,E1 -28487.488,E2 -28487.488} C_VEL
LIN {X 0,Y 72.24,Z 387.688,A -85,B 0,C 180,E1 -28494.288,E2 -28494.288} C_VEL
LIN {X 0,Y 68.996,Z 390.058,A -85,B 0,C 180,E1 -28499.383,E2 -28499.383} C_VEL
LIN {X 0,Y 66.434,Z 391.867,A -85,B 0,C 180,E1 -28504.966,E2 -28504.966} C_VEL
LIN {X 0,Y 63.226,Z 394.334,A -85,B 0,C 180,E1 -28517.155,E2 -28517.155} C_VEL
LIN {X 0,Y 62.61,Z 394.934,A -85,B 0,C 180,E1 -28523.555,E2 -28523.555} C_VEL
LIN {X 0,Y 62.581,Z 395.097,A -85,B 0,C 180,E1 -28530,E2 -28530} C_VEL
LIN {X 0,Y 62.612,Z 394.934,A -85,B 0,C 180,E1 -28536.445,E2 -28536.445} C_VEL
LIN {X 0,Y 63.233,Z 394.334,A -85,B 0,C 180,E1 -28542.843,E2 -28542.843} C_VEL
LIN {X 0,Y 66.434,Z 391.867,A -85,B 0,C 180,E1 -28555.034,E2 -28555.034} C_VEL
LIN {X 0,Y 70.562,Z 388.907,A -85,B 0,C 180,E1 -28563.216,E2 -28563.216} C_VEL
LIN {X 0,Y 75.937,Z 384.912,A -85,B 0,C 180,E1 -28570.379,E2 -28570.379} C_VEL
LIN {X 0,Y 81.656,Z 380.382,A -85,B 0,C 180,E1 -28575.894,E2 -28575.894} C_VEL
LIN {X 0,Y 88.176,Z 374.511,A -85,B 0,C 180,E1 -28580.996,E2 -28580.996} C_VEL
LIN {X 0,Y 91.905,Z 370.943,A -85,B 0,C 180,E1 -28583.41,E2 -28583.41} C_VEL
LIN {X 0,Y 95.244,Z 365.774,A -85,B 0,C 180,E1 -28587.454,E2 -28587.454} C_VEL
LIN {X 0,Y 97.814,Z 360.743,A -85,B 0,C 180,E1 -28591.24,E2 -28591.24} C_VEL
LIN {X 0,Y 98.912,Z 357.875,A -85,B 0,C 180,E1 -28593.769,E2 -28593.769} C_VEL
LIN {X 0,Y 99.32,Z 354.906,A -85,B 0,C 180,E1 -28596.908,E2 -28596.908} C_VEL
LIN {X 0,Y 99.651,Z 350.898,A -85,B 0,C 180,E1 -28602.08,E2 -28602.08} C_VEL
LIN {X 0,Y 99.826,Z 348.454,A -85,B 0,C 180,E1 -28605.712,E2 -28605.712} C_VEL
LIN {X 0,Y 99.834,Z 347.274,A -85,B 0,C 180,E1 -28607.785,E2 -28607.785} C_VEL
LIN {X 0,Y 99.673,Z 345.651,A -85,B 0,C 180,E1 -28611.87,E2 -28611.87} C_VEL
LIN {X 0,Y 99.896,Z 343.655,A -85,B 0,C 180,E1 -28619.977,E2 -28619.977} C_VEL
LIN {X 0,Y 99.337,Z 345.237,A -85,B 0,C 180,E1 -28628.11,E2 -28628.11} C_VEL
LIN {X 0,Y 99.481,Z 346.46,A -85,B 0,C 180,E1 -28632.211,E2 -28632.211} C_VEL
LIN {X 0,Y 99.792,Z 349.214,A -85,B 0,C 180,E1 -28638.451,E2 -28638.451} C_VEL
LIN {X 0,Y 100.017,Z 351.618,A -85,B 0,C 180,E1 -28642.711,E2 -28642.711} C_VEL
LIN {X 0,Y 100.127,Z 354.817,A -85,B 0,C 180,E1 -28647.117,E2 -28647.117} C_VEL
LIN {X 0,Y 100.019,Z 359.046,A -85,B 0,C 180,E1 -28652.522,E2 -28652.522} C_VEL
LIN {X 0,Y 99.489,Z 363.568,A -85,B 0,C 180,E1 -28657.581,E2 -28657.581} C_VEL
LIN {X 0,Y 98.435,Z 368.643,A -85,B 0,C 180,E1 -28663.071,E2 -28663.071} C_VEL
LIN {X 0,Y 96.931,Z 374.002,A -85,B 0,C 180,E1 -28669.267,E2 -28669.267} C_VEL
LIN {X 0,Y 96.384,Z 379.245,A -85,B 0,C 180,E1 -28676.848,E2 -28676.848} C_VEL
LIN {X 0,Y 97.791,Z 383.316,A -85,B 0,C 180,E1 -28684.457,E2 -28684.457} C_VEL
LIN {X 0,Y 99.895,Z 385.508,A -85,B 0,C 180,E1 -28689.405,E2 -28689.405} C_VEL
LIN {X 0,Y 102.961,Z 387.127,A -85,B 0,C 180,E1 -28694.155,E2 -28694.155} C_VEL
LIN {X 0,Y 111.531,Z 389.206,A -85,B 0,C 180,E1 -28702.76,E2 -28702.76} C_VEL
LIN {X 0,Y 122,Z 389.604,A -85,B 0,C 180,E1 -28709.484,E2 -28709.484} C_VEL
LIN {X 0,Y 122.972,Z 389.575,A -85,B 0,C 180,E1 -28710,E2 -28710} C_VEL
LIN {X 0,Y 114.124,Z 389.409,A -85,B 0,C 180,E1 -28715.301,E2 -28715.301} C_VEL
LIN {X 0,Y 110.262,Z 389.204,A -85,B 0,C 180,E1 -28717.591,E2 -28717.591} C_VEL
LIN {X 0,Y 97.592,Z 388.111,A -85,B 0,C 180,E1 -28724.498,E2 -28724.498} C_VEL
LIN {X 0,Y 94.51,Z 387.34,A -85,B 0,C 180,E1 -28727.446,E2 -28727.446} C_VEL
LIN {X 0,Y 93.795,Z 386.995,A -85,B 0,C 180,E1 -28728.536,E2 -28728.536} C_VEL
LIN {X 0,Y 91.632,Z 385.555,A -85,B 0,C 180,E1 -28733.092,E2 -28733.092} C_VEL
LIN {X 0,Y 89.727,Z 382.434,A -85,B 0,C 180,E1 -28740.561,E2 -28740.561} C_VEL
LIN {X 0,Y 89.801,Z 377.913,A -85,B 0,C 180,E1 -28748.762,E2 -28748.762} C_VEL
LIN {X 0,Y 91.577,Z 372.454,A -85,B 0,C 180,E1 -28756.354,E2 -28756.354} C_VEL
LIN {X 0,Y 93.275,Z 367.121,A -85,B 0,C 180,E1 -28762.965,E2 -28762.965} C_VEL
LIN {X 0,Y 94.222,Z 362.709,A -85,B 0,C 180,E1 -28768.556,E2 -28768.556} C_VEL
LIN {X 0,Y 94.543,Z 359.111,A -85,B 0,C 180,E1 -28773.541,E2 -28773.541} C_VEL
LIN {X 0,Y 94.786,Z 356.176,A -85,B 0,C 180,E1 -28778.267,E2 -28778.267} C_VEL
LIN {X 0,Y 94.764,Z 353.838,A -85,B 0,C 180,E1 -28782.77,E2 -28782.77} C_VEL
LIN {X 0,Y 94.664,Z 352.104,A -85,B 0,C 180,E1 -28787.157,E2 -28787.157} C_VEL
LIN {X 0,Y 94.716,Z 350.813,A -85,B 0,C 180,E1 -28791.491,E2 -28791.491} C_VEL
LIN {X 0,Y 95.46,Z 349.281,A -85,B 0,C 180,E1 -28800.025,E2 -28800.025} C_VEL
LIN {X 0,Y 95.018,Z 351.33,A -85,B 0,C 180,E1 -28808.531,E2 -28808.531} C_VEL
LIN {X 0,Y 94.938,Z 353.073,A -85,B 0,C 180,E1 -28812.856,E2 -28812.856} C_VEL
LIN {X 0,Y 94.27,Z 357.45,A -85,B 0,C 180,E1 -28819.627,E2 -28819.627} C_VEL
LIN {X 0,Y 93.686,Z 359.952,A -85,B 0,C 180,E1 -28822.957,E2 -28822.957} C_VEL
LIN {X 0,Y 93.141,Z 361.823,A -85,B 0,C 180,E1 -28825.117,E2 -28825.117} C_VEL
LIN {X 0,Y 91.03,Z 365.672,A -85,B 0,C 180,E1 -28828.35,E2 -28828.35} C_VEL
LIN {X 0,Y 87.576,Z 370.716,A -85,B 0,C 180,E1 -28832.583,E2 -28832.583} C_VEL
LIN {X 0,Y 86.508,Z 371.985,A -85,B 0,C 180,E1 -28833.622,E2 -28833.622} C_VEL
LIN {X 0,Y 79.285,Z 378.252,A -85,B 0,C 180,E1 -28838.387,E2 -28838.387} C_VEL
LIN {X 0,Y 72.913,Z 383.146,A -85,B 0,C 180,E1 -28843.705,E2 -28843.705} C_VEL
LIN {X 0,Y 66.591,Z 387.476,A -85,B 0,C 180,E1 -28850.711,E2 -28850.711} C_VEL
LIN {X 0,Y 62.971,Z 389.846,A -85,B 0,C 180,E1 -28856.081,E2 -28856.081} C_VEL
LIN {X 0,Y 57.817,Z 393.052,A -85,B 0,C 180,E1 -28868.613,E2 -28868.613} C_VEL
LIN {X 0,Y 56.314,Z 394.122,A -85,B 0,C 180,E1 -28875.546,E2 -28875.546} C_VEL
LIN {X 0,Y 55.564,Z 394.723,A -85,B 0,C 180,E1 -28882.734,E2 -28882.734} C_VEL
LIN {X 0,Y 55.5,Z 394.886,A -85,B 0,C 180,E1 -28890,E2 -28890} C_VEL
LIN {X 0,Y 55.566,Z 394.723,A -85,B 0,C 180,E1 -28897.266,E2 -28897.266} C_VEL
LIN {X 0,Y 56.318,Z 394.122,A -85,B 0,C 180,E1 -28904.452,E2 -28904.452} C_VEL
LIN {X 0,Y 60.034,Z 391.654,A -85,B 0,C 180,E1 -28917.921,E2 -28917.921} C_VEL
LIN {X 0,Y 64.725,Z 388.695,A -85,B 0,C 180,E1 -28926.669,E2 -28926.669} C_VEL
LIN {X 0,Y 70.659,Z 384.7,A -85,B 0,C 180,E1 -28934.126,E2 -28934.126} C_VEL
LIN {X 0,Y 76.529,Z 380.435,A -85,B 0,C 180,E1 -28939.447,E2 -28939.447} C_VEL
LIN {X 0,Y 82.572,Z 375.455,A -85,B 0,C 180,E1 -28943.956,E2 -28943.956} C_VEL
LIN {X 0,Y 86.496,Z 371.985,A -85,B 0,C 180,E1 -28946.389,E2 -28946.389} C_VEL
LIN {X 0,Y 90.281,Z 366.783,A -85,B 0,C 180,E1 -28950.69,E2 -28950.69} C_VEL
LIN {X 0,Y 92.596,Z 362.977,A -85,B 0,C 180,E1 -28953.858,E2 -28953.858} C_VEL
LIN {X 0,Y 93.132,Z 361.822,A -85,B 0,C 180,E1 -28954.896,E2 -28954.896} C_VEL
LIN {X 0,Y 93.901,Z 359.177,A -85,B 0,C 180,E1 -28957.998,E2 -28957.998} C_VEL
LIN {X 0,Y 94.507,Z 355.831,A -85,B 0,C 180,E1 -28962.67,E2 -28962.67} C_VEL
LIN {X 0,Y 94.952,Z 353.058,A -85,B 0,C 180,E1 -28967.146,E2 -28967.146} C_VEL
LIN {X 0,Y 95.074,Z 351.269,A -85,B 0,C 180,E1 -28971.474,E2 -28971.474} C_VEL
LIN {X 0,Y 95.455,Z 349.287,A -85,B 0,C 180,E1 -28979.975,E2 -28979.975} C_VEL
LIN {X 0,Y 94.719,Z 350.81,A -85,B 0,C 180,E1 -28988.509,E2 -28988.509} C_VEL
LIN {X 0,Y 94.717,Z 353.003,A -85,B 0,C 180,E1 -28995.296,E2 -28995.296} C_VEL
LIN {X 0,Y 94.831,Z 354.923,A -85,B 0,C 180,E1 -28999.454,E2 -28999.454} C_VEL
LIN {X 0,Y 94.703,Z 357.523,A -85,B 0,C 180,E1 -29004.06,E2 -29004.06} C_VEL
LIN {X 0,Y 94.407,Z 360.847,A -85,B 0,C 180,E1 -29008.907,E2 -29008.907} C_VEL
LIN {X 0,Y 94.012,Z 363.764,A -85,B 0,C 180,E1 -29012.87,E2 -29012.87} C_VEL
LIN {X 0,Y 93.019,Z 368.181,A -85,B 0,C 180,E1 -29018.29,E2 -29018.29} C_VEL
LIN {X 0,Y 91.573,Z 372.457,A -85,B 0,C 180,E1 -29023.649,E2 -29023.649} C_VEL
LIN {X 0,Y 89.791,Z 378.058,A -85,B 0,C 180,E1 -29031.462,E2 -29031.462} C_VEL
LIN {X 0,Y 89.713,Z 382.445,A -85,B 0,C 180,E1 -29039.454,E2 -29039.454} C_VEL
LIN {X 0,Y 91.754,Z 385.769,A -85,B 0,C 180,E1 -29047.482,E2 -29047.482} C_VEL
LIN {X 0,Y 95.125,Z 387.729,A -85,B 0,C 180,E1 -29053.735,E2 -29053.735} C_VEL
LIN {X 0,Y 102.39,Z 389.481,A -85,B 0,C 180,E1 -29062.11,E2 -29062.11} C_VEL
LIN {X 0,Y 107.552,Z 389.888,A -85,B 0,C 180,E1 -29066.253,E2 -29066.253} C_VEL
LIN {X 0,Y 113.483,Z 389.857,A -85,B 0,C 180,E1 -29070,E2 -29070} C_VEL
LIN {X 0,Y 105.783,Z 389.757,A -85,B 0,C 180,E1 -29075.047,E2 -29075.047} C_VEL
LIN {X 0,Y 99.94,Z 389.074,A -85,B 0,C 180,E1 -29080.251,E2 -29080.251} C_VEL
LIN {X 0,Y 93.795,Z 386.995,A -85,B 0,C 180,E1 -29088.536,E2 -29088.536} C_VEL
LIN {X 0,Y 91.496,Z 386.053,A -85,B 0,C 180,E1 -29091.853,E2 -29091.853} C_VEL
LIN {X 0,Y 83.77,Z 382.989,A -85,B 0,C 180,E1 -29102.184,E2 -29102.184} C_VEL
LIN {X 0,Y 82.728,Z 381.448,A -85,B 0,C 180,E1 -29106.011,E2 -29106.011} C_VEL
LIN {X 0,Y 82.742,Z 380.818,A -85,B 0,C 180,E1 -29107.296,E2 -29107.296} C_VEL
LIN {X 0,Y 84.33,Z 376.321,A -85,B 0,C 180,E1 -29115.102,E2 -29115.102} C_VEL
LIN {X 0,Y 86.106,Z 372.345,A -85,B 0,C 180,E1 -29120.917,E2 -29120.917} C_VEL
LIN {X 0,Y 87.488,Z 368.872,A -85,B 0,C 180,E1 -29125.819,E2 -29125.819} C_VEL
LIN {X 0,Y 88.419,Z 365.295,A -85,B 0,C 180,E1 -29130.965,E2 -29130.965} C_VEL
LIN {X 0,Y 89.184,Z 361.767,A -85,B 0,C 180,E1 -29136.825,E2 -29136.825} C_VEL
LIN {X 0,Y 89.462,Z 359.248,A -85,B 0,C 180,E1 -29141.714,E2 -29141.714} C_VEL
LIN {X 0,Y 89.603,Z 357.471,A -85,B 0,C 180,E1 -29146.418,E2 -29146.418} C_VEL
LIN {X 0,Y 89.792,Z 356.191,A -85,B 0,C 180,E1 -29151.021,E2 -29151.021} C_VEL
LIN {X 0,Y 90.604,Z 354.573,A -85,B 0,C 180,E1 -29160.026,E2 -29160.026} C_VEL
LIN {X 0,Y 90.189,Z 355.537,A -85,B 0,C 180,E1 -29164.495,E2 -29164.495} C_VEL
LIN {X 0,Y 90.038,Z 356.793,A -85,B 0,C 180,E1 -29169.007,E2 -29169.007} C_VEL
LIN {X 0,Y 89.599,Z 358.748,A -85,B 0,C 180,E1 -29173.636,E2 -29173.636} C_VEL
LIN {X 0,Y 88.777,Z 361.613,A -85,B 0,C 180,E1 -29178.488,E2 -29178.488} C_VEL
LIN {X 0,Y 87.886,Z 364.433,A -85,B 0,C 180,E1 -29182.352,E2 -29182.352} C_VEL
LIN {X 0,Y 87.138,Z 365.737,A -85,B 0,C 180,E1 -29183.81,E2 -29183.81} C_VEL
LIN {X 0,Y 83.631,Z 370.484,A -85,B 0,C 180,E1 -29188.072,E2 -29188.072} C_VEL
LIN {X 0,Y 81.355,Z 372.929,A -85,B 0,C 180,E1 -29190.248,E2 -29190.248} C_VEL
LIN {X 0,Y 74.328,Z 378.565,A -85,B 0,C 180,E1 -29194.599,E2 -29194.599} C_VEL
LIN {X 0,Y 68.189,Z 382.934,A -85,B 0,C 180,E1 -29199.378,E2 -29199.378} C_VEL
LIN {X 0,Y 61.248,Z 387.264,A -85,B 0,C 180,E1 -29206.491,E2 -29206.491} C_VEL
LIN {X 0,Y 57.204,Z 389.635,A -85,B 0,C 180,E1 -29212.101,E2 -29212.101} C_VEL
LIN {X 0,Y 51.231,Z 392.84,A -85,B 0,C 180,E1 -29225.699,E2 -29225.699} C_VEL
LIN {X 0,Y 49.438,Z 393.91,A -85,B 0,C 180,E1 -29233.483,E2 -29233.483} C_VEL
LIN {X 0,Y 48.521,Z 394.511,A -85,B 0,C 180,E1 -29241.672,E2 -29241.672} C_VEL
LIN {X 0,Y 48.401,Z 394.675,A -85,B 0,C 180,E1 -29250,E2 -29250} C_VEL
LIN {X 0,Y 48.524,Z 394.511,A -85,B 0,C 180,E1 -29258.328,E2 -29258.328} C_VEL
LIN {X 0,Y 49.443,Z 393.91,A -85,B 0,C 180,E1 -29266.516,E2 -29266.516} C_VEL
LIN {X 0,Y 53.826,Z 391.441,A -85,B 0,C 180,E1 -29281.484,E2 -29281.484} C_VEL
LIN {X 0,Y 59.173,Z 388.483,A -85,B 0,C 180,E1 -29290.785,E2 -29290.785} C_VEL
LIN {X 0,Y 65.734,Z 384.488,A -85,B 0,C 180,E1 -29298.452,E2 -29298.452} C_VEL
LIN {X 0,Y 72.766,Z 379.696,A -85,B 0,C 180,E1 -29304.321,E2 -29304.321} C_VEL
LIN {X 0,Y 79.959,Z 374.086,A -85,B 0,C 180,E1 -29308.977,E2 -29308.977} C_VEL
LIN {X 0,Y 81.354,Z 372.929,A -85,B 0,C 180,E1 -29309.753,E2 -29309.753} C_VEL
LIN {X 0,Y 84.675,Z 369.08,A -85,B 0,C 180,E1 -29313.155,E2 -29313.155} C_VEL
LIN {X 0,Y 87.167,Z 365.712,A -85,B 0,C 180,E1 -29316.198,E2 -29316.198} C_VEL
LIN {X 0,Y 88.274,Z 363.374,A -85,B 0,C 180,E1 -29318.979,E2 -29318.979} C_VEL
LIN {X 0,Y 89.192,Z 360.174,A -85,B 0,C 180,E1 -29323.797,E2 -29323.797} C_VEL
LIN {X 0,Y 89.94,Z 357.605,A -85,B 0,C 180,E1 -29328.709,E2 -29328.709} C_VEL
LIN {X 0,Y 90.076,Z 356.753,A -85,B 0,C 180,E1 -29330.997,E2 -29330.997} C_VEL
LIN {X 0,Y 90.223,Z 355.5,A -85,B 0,C 180,E1 -29335.507,E2 -29335.507} C_VEL
LIN {X 0,Y 90.615,Z 354.562,A -85,B 0,C 180,E1 -29339.974,E2 -29339.974} C_VEL
LIN {X 0,Y 89.793,Z 356.19,A -85,B 0,C 180,E1 -29348.979,E2 -29348.979} C_VEL
LIN {X 0,Y 89.614,Z 357.461,A -85,B 0,C 180,E1 -29353.58,E2 -29353.58} C_VEL
LIN {X 0,Y 89.411,Z 359.762,A -85,B 0,C 180,E1 -29359.4,E2 -29359.4} C_VEL
LIN {X 0,Y 88.968,Z 362.874,A -85,B 0,C 180,E1 -29365.033,E2 -29365.033} C_VEL
LIN {X 0,Y 88.106,Z 366.727,A -85,B 0,C 180,E1 -29371.195,E2 -29371.195} C_VEL
LIN {X 0,Y 86.975,Z 370.184,A -85,B 0,C 180,E1 -29376.096,E2 -29376.096} C_VEL
LIN {X 0,Y 85.212,Z 374.488,A -85,B 0,C 180,E1 -29382.075,E2 -29382.075} C_VEL
LIN {X 0,Y 82.907,Z 380.172,A -85,B 0,C 180,E1 -29391.444,E2 -29391.444} C_VEL
LIN {X 0,Y 82.764,Z 383.822,A -85,B 0,C 180,E1 -29399.37,E2 -29399.37} C_VEL
LIN {X 0,Y 84.285,Z 386.363,A -85,B 0,C 180,E1 -29406.445,E2 -29406.445} C_VEL
LIN {X 0,Y 87.706,Z 388.414,A -85,B 0,C 180,E1 -29413.956,E2 -29413.956} C_VEL
LIN {X 0,Y 93.384,Z 389.752,A -85,B 0,C 180,E1 -29421.343,E2 -29421.343} C_VEL
LIN {X 0,Y 98.577,Z 390.178,A -85,B 0,C 180,E1 -29426.069,E2 -29426.069} C_VEL
LIN {X 0,Y 104.042,Z 390.138,A -85,B 0,C 180,E1 -29430,E2 -29430} C_VEL
LIN {X 0,Y 98.321,Z 390.164,A -85,B 0,C 180,E1 -29434.099,E2 -29434.099} C_VEL
LIN {X 0,Y 92.596,Z 389.662,A -85,B 0,C 180,E1 -29439.531,E2 -29439.531} C_VEL
LIN {X 0,Y 86.187,Z 387.65,A -85,B 0,C 180,E1 -29449.036,E2 -29449.036} C_VEL
LIN {X 0,Y 83.257,Z 384.955,A -85,B 0,C 180,E1 -29457.662,E2 -29457.662} C_VEL
LIN {X 0,Y 82.676,Z 381.213,A -85,B 0,C 180,E1 -29466.515,E2 -29466.515} C_VEL
LIN {X 0,Y 82.742,Z 380.818,A -85,B 0,C 180,E1 -29467.296,E2 -29467.296} C_VEL
LIN {X 0,Y 82.692,Z 379.026,A -85,B 0,C 180,E1 -29471.19,E2 -29471.19} C_VEL
LIN {X 0,Y 81.649,Z 376.113,A -85,B 0,C 180,E1 -29477.777,E2 -29477.777} C_VEL
LIN {X 0,Y 81.114,Z 372.442,A -85,B 0,C 180,E1 -29485.838,E2 -29485.838} C_VEL
LIN {X 0,Y 81.61,Z 370.924,A -85,B 0,C 180,E1 -29488.435,E2 -29488.435} C_VEL
LIN {X 0,Y 82.662,Z 368.338,A -85,B 0,C 180,E1 -29492.927,E2 -29492.927} C_VEL
LIN {X 0,Y 83.441,Z 365.638,A -85,B 0,C 180,E1 -29497.893,E2 -29497.893} C_VEL
LIN {X 0,Y 83.775,Z 364.469,A -85,B 0,C 180,E1 -29500.424,E2 -29500.424} C_VEL
LIN {X 0,Y 84.151,Z 362.643,A -85,B 0,C 180,E1 -29505.52,E2 -29505.52} C_VEL
LIN {X 0,Y 84.452,Z 361.201,A -85,B 0,C 180,E1 -29510.448,E2 -29510.448} C_VEL
LIN {X 0,Y 85.482,Z 359.589,A -85,B 0,C 180,E1 -29520.027,E2 -29520.027} C_VEL
LIN {X 0,Y 84.833,Z 360.92,A -85,B 0,C 180,E1 -29526.215,E2 -29526.215} C_VEL
LIN {X 0,Y 84.296,Z 362.922,A -85,B 0,C 180,E1 -29532.058,E2 -29532.058} C_VEL
LIN {X 0,Y 83.853,Z 364.181,A -85,B 0,C 180,E1 -29534.591,E2 -29534.591} C_VEL
LIN {X 0,Y 82.333,Z 367.416,A -85,B 0,C 180,E1 -29540.125,E2 -29540.125} C_VEL
LIN {X 0,Y 81.557,Z 368.519,A -85,B 0,C 180,E1 -29541.379,E2 -29541.379} C_VEL
LIN {X 0,Y 77.843,Z 372.706,A -85,B 0,C 180,E1 -29545.468,E2 -29545.468} C_VEL
LIN {X 0,Y 75.062,Z 375.03,A -85,B 0,C 180,E1 -29547.195,E2 -29547.195} C_VEL
LIN {X 0,Y 66.604,Z 381.06,A -85,B 0,C 180,E1 -29552.42,E2 -29552.42} C_VEL
LIN {X 0,Y 58.696,Z 385.808,A -85,B 0,C 180,E1 -29558.897,E2 -29558.897} C_VEL
LIN {X 0,Y 51.779,Z 389.423,A -85,B 0,C 180,E1 -29567.262,E2 -29567.262} C_VEL
LIN {X 0,Y 47.882,Z 391.229,A -85,B 0,C 180,E1 -29574.049,E2 -29574.049} C_VEL
LIN {X 0,Y 42.656,Z 393.698,A -85,B 0,C 180,E1 -29590.761,E2 -29590.761} C_VEL
LIN {X 0,Y 41.493,Z 394.299,A -85,B 0,C 180,E1 -29600.249,E2 -29600.249} C_VEL
LIN {X 0,Y 41.317,Z 394.464,A -85,B 0,C 180,E1 -29610,E2 -29610} C_VEL
LIN {X 0,Y 41.495,Z 394.299,A -85,B 0,C 180,E1 -29619.751,E2 -29619.751} C_VEL
LIN {X 0,Y 42.659,Z 393.698,A -85,B 0,C 180,E1 -29629.238,E2 -29629.238} C_VEL
LIN {X 0,Y 47.882,Z 391.229,A -85,B 0,C 180,E1 -29645.952,E2 -29645.952} C_VEL
LIN {X 0,Y 53.97,Z 388.271,A -85,B 0,C 180,E1 -29655.742,E2 -29655.742} C_VEL
LIN {X 0,Y 61.246,Z 384.276,A -85,B 0,C 180,E1 -29663.441,E2 -29663.441} C_VEL
LIN {X 0,Y 68.084,Z 380.007,A -85,B 0,C 180,E1 -29668.659,E2 -29668.659} C_VEL
LIN {X 0,Y 75.058,Z 375.03,A -85,B 0,C 180,E1 -29672.811,E2 -29672.811} C_VEL
LIN {X 0,Y 76.525,Z 373.873,A -85,B 0,C 180,E1 -29673.562,E2 -29673.562} C_VEL
LIN {X 0,Y 79.012,Z 371.526,A -85,B 0,C 180,E1 -29675.742,E2 -29675.742} C_VEL
LIN {X 0,Y 81.565,Z 368.519,A -85,B 0,C 180,E1 -29678.607,E2 -29678.607} C_VEL
LIN {X 0,Y 82.36,Z 367.338,A -85,B 0,C 180,E1 -29680.013,E2 -29680.013} C_VEL
LIN {X 0,Y 83.853,Z 364.182,A -85,B 0,C 180,E1 -29685.409,E2 -29685.409} C_VEL
LIN {X 0,Y 84.681,Z 361.836,A -85,B 0,C 180,E1 -29690.418,E2 -29690.418} C_VEL
LIN {X 0,Y 84.984,Z 360.529,A -85,B 0,C 180,E1 -29695.229,E2 -29695.229} C_VEL
LIN {X 0,Y 85.481,Z 359.59,A -85,B 0,C 180,E1 -29699.973,E2 -29699.973} C_VEL
LIN {X 0,Y 84.453,Z 361.2,A -85,B 0,C 180,E1 -29709.552,E2 -29709.552} C_VEL
LIN {X 0,Y 84.161,Z 362.634,A -85,B 0,C 180,E1 -29714.479,E2 -29714.479} C_VEL
LIN {X 0,Y 83.807,Z 364.443,A -85,B 0,C 180,E1 -29719.568,E2 -29719.568} C_VEL
LIN {X 0,Y 82.957,Z 367.197,A -85,B 0,C 180,E1 -29725.029,E2 -29725.029} C_VEL
LIN {X 0,Y 81.817,Z 370.463,A -85,B 0,C 180,E1 -29730.798,E2 -29730.798} C_VEL
LIN {X 0,Y 80.35,Z 373.752,A -85,B 0,C 180,E1 -29735.996,E2 -29735.996} C_VEL
LIN {X 0,Y 77.736,Z 378.399,A -85,B 0,C 180,E1 -29743.676,E2 -29743.676} C_VEL
LIN {X 0,Y 75.883,Z 382.907,A -85,B 0,C 180,E1 -29752.987,E2 -29752.987} C_VEL
LIN {X 0,Y 76.26,Z 386.277,A -85,B 0,C 180,E1 -29762.562,E2 -29762.562} C_VEL
LIN {X 0,Y 77.916,Z 387.912,A -85,B 0,C 180,E1 -29768.851,E2 -29768.851} C_VEL
LIN {X 0,Y 80.672,Z 389.133,A -85,B 0,C 180,E1 -29774.85,E2 -29774.85} C_VEL
LIN {X 0,Y 85.266,Z 390.089,A -85,B 0,C 180,E1 -29781.322,E2 -29781.322} C_VEL
LIN {X 0,Y 91.411,Z 390.517,A -85,B 0,C 180,E1 -29787.405,E2 -29787.405} C_VEL
LIN {X 0,Y 94.744,Z 390.415,A -85,B 0,C 180,E1 -29790,E2 -29790} C_VEL
LIN {X 0,Y 89.218,Z 390.435,A -85,B 0,C 180,E1 -29794.518,E2 -29794.518} C_VEL
LIN {X 0,Y 84.543,Z 390.018,A -85,B 0,C 180,E1 -29799.57,E2 -29799.57} C_VEL
LIN {X 0,Y 77.986,Z 387.91,A -85,B 0,C 180,E1 -29811.129,E2 -29811.129} C_VEL
LIN {X 0,Y 75.85,Z 385.297,A -85,B 0,C 180,E1 -29820.398,E2 -29820.398} C_VEL
LIN {X 0,Y 76.22,Z 381.457,A -85,B 0,C 180,E1 -29830.198,E2 -29830.198} C_VEL
LIN {X 0,Y 78.644,Z 376.726,A -85,B 0,C 180,E1 -29839.084,E2 -29839.084} C_VEL
LIN {X 0,Y 80.847,Z 372.652,A -85,B 0,C 180,E1 -29845.672,E2 -29845.672} C_VEL
LIN {X 0,Y 81.61,Z 370.924,A -85,B 0,C 180,E1 -29848.435,E2 -29848.435} C_VEL
LIN {X 0,Y 81.989,Z 369.59,A -85,B 0,C 180,E1 -29851,E2 -29851} C_VEL
LIN {X 0,Y 81.631,Z 368.17,A -85,B 0,C 180,E1 -29855.021,E2 -29855.021} C_VEL
LIN {X 0,Y 80.678,Z 367.305,A -85,B 0,C 180,E1 -29859.148,E2 -29859.148} C_VEL
LIN {X 0,Y 78.877,Z 365.739,A -85,B 0,C 180,E1 -29870.991,E2 -29870.991} C_VEL
LIN {X 0,Y 79.367,Z 364.998,A -85,B 0,C 180,E1 -29874.95,E2 -29874.95} C_VEL
LIN {X 0,Y 80.106,Z 364.391,A -85,B 0,C 180,E1 -29880.029,E2 -29880.029} C_VEL
LIN {X 0,Y 79.489,Z 365.327,A -85,B 0,C 180,E1 -29885.102,E2 -29885.102} C_VEL
LIN {X 0,Y 78.72,Z 367.015,A -85,B 0,C 180,E1 -29890.875,E2 -29890.875} C_VEL
LIN {X 0,Y 77.438,Z 369.389,A -85,B 0,C 180,E1 -29895.83,E2 -29895.83} C_VEL
LIN {X 0,Y 76.857,Z 370.425,A -85,B 0,C 180,E1 -29897.654,E2 -29897.654} C_VEL
LIN {X 0,Y 73.491,Z 373.65,A -85,B 0,C 180,E1 -29901.191,E2 -29901.191} C_VEL
LIN {X 0,Y 70.546,Z 375.973,A -85,B 0,C 180,E1 -29902.854,E2 -29902.854} C_VEL
LIN {X 0,Y 60.161,Z 382.51,A -85,B 0,C 180,E1 -29908.821,E2 -29908.821} C_VEL
LIN {X 0,Y 51.827,Z 386.839,A -85,B 0,C 180,E1 -29915.549,E2 -29915.549} C_VEL
LIN {X 0,Y 46.805,Z 389.211,A -85,B 0,C 180,E1 -29921.344,E2 -29921.344} C_VEL
LIN {X 0,Y 42.312,Z 391.016,A -85,B 0,C 180,E1 -29928.365,E2 -29928.365} C_VEL
LIN {X 0,Y 36.014,Z 393.486,A -85,B 0,C 180,E1 -29947.028,E2 -29947.028} C_VEL
LIN {X 0,Y 34.514,Z 394.088,A -85,B 0,C 180,E1 -29958.251,E2 -29958.251} C_VEL
LIN {X 0,Y 34.208,Z 394.253,A -85,B 0,C 180,E1 -29970,E2 -29970} C_VEL
LIN {X 0,Y 34.516,Z 394.088,A -85,B 0,C 180,E1 -29981.748,E2 -29981.748} C_VEL
LIN {X 0,Y 36.017,Z 393.486,A -85,B 0,C 180,E1 -29992.971,E2 -29992.971} C_VEL
LIN {X 0,Y 42.312,Z 391.016,A -85,B 0,C 180,E1 -30011.635,E2 -30011.635} C_VEL
LIN {X 0,Y 49.257,Z 388.058,A -85,B 0,C 180,E1 -30021.695,E2 -30021.695} C_VEL
LIN {X 0,Y 57.294,Z 384.064,A -85,B 0,C 180,E1 -30029.164,E2 -30029.164} C_VEL
LIN {X 0,Y 65.854,Z 379.04,A -85,B 0,C 180,E1 -30034.692,E2 -30034.692} C_VEL
LIN {X 0,Y 72.082,Z 374.818,A -85,B 0,C 180,E1 -30037.854,E2 -30037.854} C_VEL
LIN {X 0,Y 74.765,Z 372.469,A -85,B 0,C 180,E1 -30040.05,E2 -30040.05} C_VEL
LIN {X 0,Y 76.846,Z 370.436,A -85,B 0,C 180,E1 -30042.336,E2 -30042.336} C_VEL
LIN {X 0,Y 78.32,Z 367.797,A -85,B 0,C 180,E1 -30047.27,E2 -30047.27} C_VEL
LIN {X 0,Y 78.886,Z 366.75,A -85,B 0,C 180,E1 -30049.707,E2 -30049.707} C_VEL
LIN {X 0,Y 79.518,Z 365.304,A -85,B 0,C 180,E1 -30054.9,E2 -30054.9} C_VEL
LIN {X 0,Y 80.109,Z 364.388,A -85,B 0,C 180,E1 -30059.971,E2 -30059.971} C_VEL
LIN {X 0,Y 79.054,Z 365.401,A -85,B 0,C 180,E1 -30067.198,E2 -30067.198} C_VEL
LIN {X 0,Y 78.723,Z 366.13,A -85,B 0,C 180,E1 -30070.885,E2 -30070.885} C_VEL
LIN {X 0,Y 78.082,Z 368.326,A -85,B 0,C 180,E1 -30078.33,E2 -30078.33} C_VEL
LIN {X 0,Y 76.946,Z 370.777,A -85,B 0,C 180,E1 -30084.027,E2 -30084.027} C_VEL
LIN {X 0,Y 75.564,Z 373.652,A -85,B 0,C 180,E1 -30089.751,E2 -30089.751} C_VEL
LIN {X 0,Y 73.873,Z 376.325,A -85,B 0,C 180,E1 -30094.766,E2 -30094.766} C_VEL
LIN {X 0,Y 71.229,Z 380.115,A -85,B 0,C 180,E1 -30101.959,E2 -30101.959} C_VEL
LIN {X 0,Y 68.994,Z 384.317,A -85,B 0,C 180,E1 -30112.326,E2 -30112.326} C_VEL
LIN {X 0,Y 68.864,Z 386.529,A -85,B 0,C 180,E1 -30119.318,E2 -30119.318} C_VEL
LIN {X 0,Y 69.935,Z 388.169,A -85,B 0,C 180,E1 -30126.299,E2 -30126.299} C_VEL
LIN {X 0,Y 75.725,Z 390.285,A -85,B 0,C 180,E1 -30139.303,E2 -30139.303} C_VEL
LIN {X 0,Y 84.304,Z 390.726,A -85,B 0,C 180,E1 -30148.962,E2 -30148.962} C_VEL
LIN {X 0,Y 85.509,Z 390.69,A -85,B 0,C 180,E1 -30150,E2 -30150} C_VEL
LIN {X 0,Y 77.957,Z 390.505,A -85,B 0,C 180,E1 -30157.654,E2 -30157.654} C_VEL
LIN {X 0,Y 72.356,Z 389.39,A -85,B 0,C 180,E1 -30166.941,E2 -30166.941} C_VEL
LIN {X 0,Y 69.725,Z 387.858,A -85,B 0,C 180,E1 -30174.972,E2 -30174.972} C_VEL
LIN {X 0,Y 68.863,Z 386.529,A -85,B 0,C 180,E1 -30180.682,E2 -30180.682} C_VEL
LIN {X 0,Y 69.428,Z 383.155,A -85,B 0,C 180,E1 -30191.145,E2 -30191.145} C_VEL
LIN {X 0,Y 72.327,Z 378.643,A -85,B 0,C 180,E1 -30201.018,E2 -30201.018} C_VEL
LIN {X 0,Y 74.783,Z 375,A -85,B 0,C 180,E1 -30207.756,E2 -30207.756} C_VEL
LIN {X 0,Y 76.198,Z 372.396,A -85,B 0,C 180,E1 -30212.574,E2 -30212.574} C_VEL
LIN {X 0,Y 77.57,Z 369.542,A -85,B 0,C 180,E1 -30218.786,E2 -30218.786} C_VEL
LIN {X 0,Y 78.053,Z 368.35,A -85,B 0,C 180,E1 -30221.663,E2 -30221.663} C_VEL
LIN {X 0,Y 78.802,Z 365.969,A -85,B 0,C 180,E1 -30229.756,E2 -30229.756} C_VEL
LIN {X 0,Y 78.877,Z 365.739,A -85,B 0,C 180,E1 -30230.991,E2 -30230.991} C_VEL
LIN {X 0,Y 78.601,Z 365.682,A -85,B 0,C 180,E1 -30233.823,E2 -30233.823} C_VEL
LIN {X 0,Y 77.648,Z 366.318,A -85,B 0,C 180,E1 -30236.607,E2 -30236.607} C_VEL
LIN {X 0,Y 73.472,Z 370.095,A -85,B 0,C 180,E1 -30246.191,E2 -30246.191} C_VEL
LIN {X 0,Y 72.57,Z 371.534,A -85,B 0,C 180,E1 -30251.2,E2 -30251.2} C_VEL
LIN {X 0,Y 71.543,Z 372.846,A -85,B 0,C 180,E1 -30254.246,E2 -30254.246} C_VEL
LIN {X 0,Y 69.587,Z 374.593,A -85,B 0,C 180,E1 -30256.373,E2 -30256.373} C_VEL
LIN {X 0,Y 66.485,Z 376.797,A -85,B 0,C 180,E1 -30257.944,E2 -30257.944} C_VEL
LIN {X 0,Y 57.061,Z 382.297,A -85,B 0,C 180,E1 -30262.523,E2 -30262.523} C_VEL
LIN {X 0,Y 48.025,Z 386.626,A -85,B 0,C 180,E1 -30268.594,E2 -30268.594} C_VEL
